REGION Network 7: Choose Flush Destination
   // #Cmd.Flush_Select.%X0 = T-20.00
   // #Cmd.Flush_Select.%X1 = T-21.00
   // #Cmd.Flush_Select.%X2 = T-30.00
   // #Cmd.Flush_Select.%X3 = T-31.00
   // #Cmd.Flush_Select.%X4 = Drain
   // #Cmd.Flush_Select.%X5 = Flush_Selected
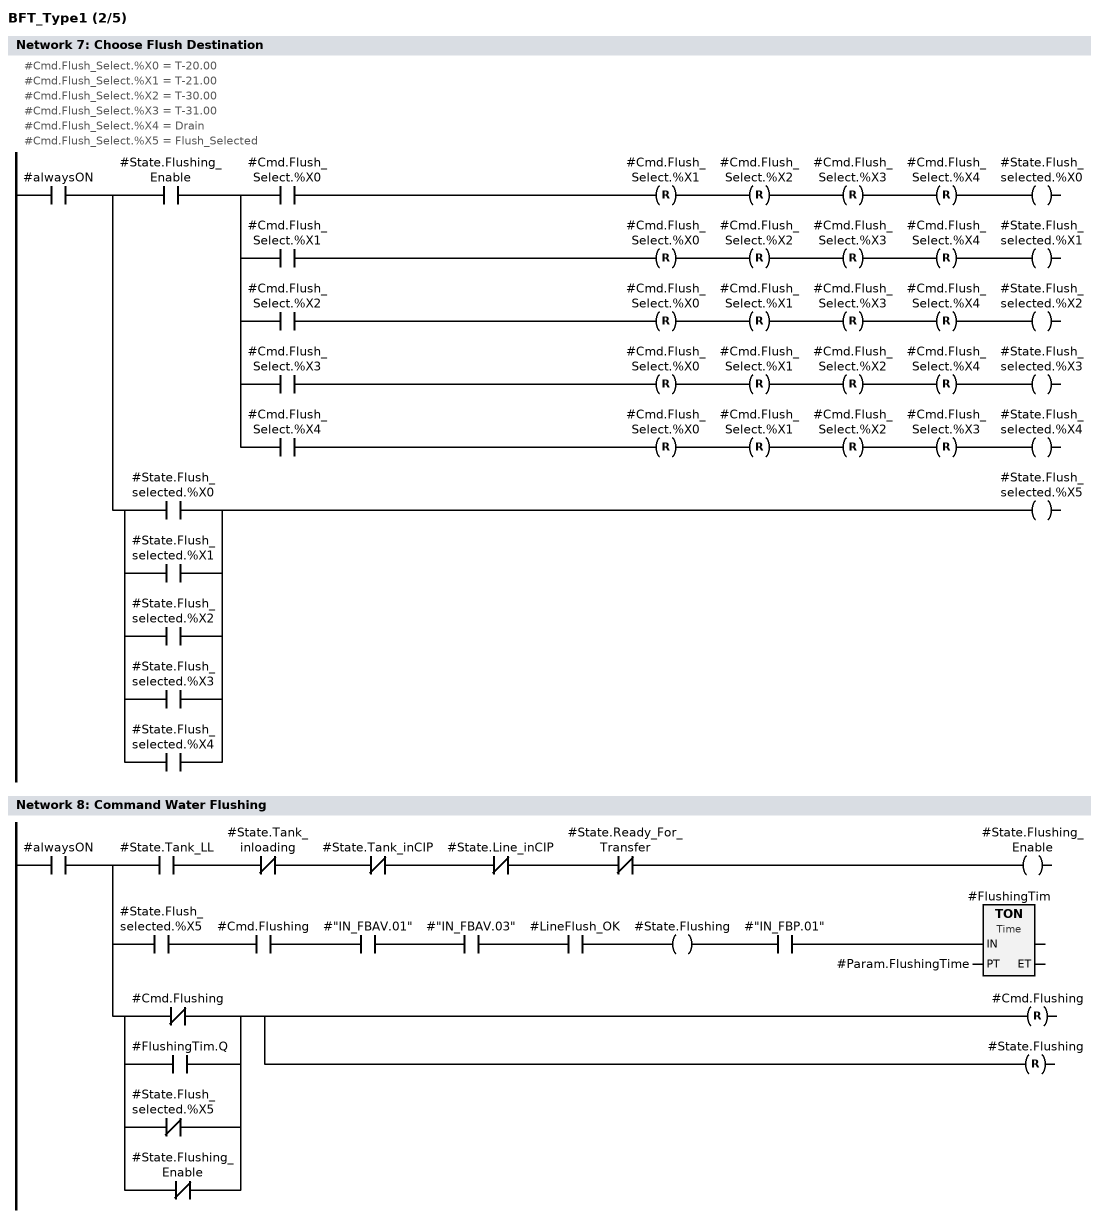
   RUNG wire#powerrail
      Contact( #alwaysON )
      wire#w1
      Contact( #State.Flushing_Enable )
      wire#w2
      Contact( #Cmd.Flush_Select.%X0 )
      R_Coil( #Cmd.Flush_Select.%X1 )
      R_Coil( #Cmd.Flush_Select.%X2 )
      R_Coil( #Cmd.Flush_Select.%X3 )
      R_Coil( #Cmd.Flush_Select.%X4 )
      Coil( #State.Flush_selected.%X0 )
   END_RUNG
   RUNG wire#w2
      Contact( #Cmd.Flush_Select.%X1 )
      R_Coil( #Cmd.Flush_Select.%X0 )
      R_Coil( #Cmd.Flush_Select.%X2 )
      R_Coil( #Cmd.Flush_Select.%X3 )
      R_Coil( #Cmd.Flush_Select.%X4 )
      Coil( #State.Flush_selected.%X1 )
   END_RUNG
   RUNG wire#w2
      Contact( #Cmd.Flush_Select.%X2 )
      R_Coil( #Cmd.Flush_Select.%X0 )
      R_Coil( #Cmd.Flush_Select.%X1 )
      R_Coil( #Cmd.Flush_Select.%X3 )
      R_Coil( #Cmd.Flush_Select.%X4 )
      Coil( #State.Flush_selected.%X2 )
   END_RUNG
   RUNG wire#w2
      Contact( #Cmd.Flush_Select.%X3 )
      R_Coil( #Cmd.Flush_Select.%X0 )
      R_Coil( #Cmd.Flush_Select.%X1 )
      R_Coil( #Cmd.Flush_Select.%X2 )
      R_Coil( #Cmd.Flush_Select.%X4 )
      Coil( #State.Flush_selected.%X3 )
   END_RUNG
   RUNG wire#w2
      Contact( #Cmd.Flush_Select.%X4 )
      R_Coil( #Cmd.Flush_Select.%X0 )
      R_Coil( #Cmd.Flush_Select.%X1 )
      R_Coil( #Cmd.Flush_Select.%X2 )
      R_Coil( #Cmd.Flush_Select.%X3 )
      Coil( #State.Flush_selected.%X4 )
   END_RUNG
   RUNG wire#w1
      Contact( #State.Flush_selected.%X0 )
      wire#w3
      Coil( #State.Flush_selected.%X5 )
   END_RUNG
   RUNG wire#w1
      Contact( #State.Flush_selected.%X1 )
   END_RUNG wire#w3
   RUNG wire#w1
      Contact( #State.Flush_selected.%X2 )
   END_RUNG wire#w3
   RUNG wire#w1
      Contact( #State.Flush_selected.%X3 )
   END_RUNG wire#w3
   RUNG wire#w1
      Contact( #State.Flush_selected.%X4 )
   END_RUNG wire#w3
   // the same network as SCL:
   #_w1 := #alwaysON AND #State.Flushing_Enable;
   #_w2 := #_w1 AND #Cmd.Flush_Select.%X0;
   IF #_w2 THEN
       #Cmd.Flush_Select.%X1 := FALSE;
       #Cmd.Flush_Select.%X2 := FALSE;
       #Cmd.Flush_Select.%X3 := FALSE;
       #Cmd.Flush_Select.%X4 := FALSE;
   END_IF;
   #State.Flush_selected.%X0 := #_w2;
   #_w3 := #_w1 AND #Cmd.Flush_Select.%X1;
   IF #_w3 THEN
       #Cmd.Flush_Select.%X0 := FALSE;
       #Cmd.Flush_Select.%X2 := FALSE;
       #Cmd.Flush_Select.%X3 := FALSE;
       #Cmd.Flush_Select.%X4 := FALSE;
   END_IF;
   #State.Flush_selected.%X1 := #_w3;
   #_w4 := #_w1 AND #Cmd.Flush_Select.%X2;
   IF #_w4 THEN
       #Cmd.Flush_Select.%X0 := FALSE;
       #Cmd.Flush_Select.%X1 := FALSE;
       #Cmd.Flush_Select.%X3 := FALSE;
       #Cmd.Flush_Select.%X4 := FALSE;
   END_IF;
   #State.Flush_selected.%X2 := #_w4;
   #_w5 := #_w1 AND #Cmd.Flush_Select.%X3;
   IF #_w5 THEN
       #Cmd.Flush_Select.%X0 := FALSE;
       #Cmd.Flush_Select.%X1 := FALSE;
       #Cmd.Flush_Select.%X2 := FALSE;
       #Cmd.Flush_Select.%X4 := FALSE;
   END_IF;
   #State.Flush_selected.%X3 := #_w5;
   #_w6 := #_w1 AND #Cmd.Flush_Select.%X4;
   IF #_w6 THEN
       #Cmd.Flush_Select.%X0 := FALSE;
       #Cmd.Flush_Select.%X1 := FALSE;
       #Cmd.Flush_Select.%X2 := FALSE;
       #Cmd.Flush_Select.%X3 := FALSE;
   END_IF;
   #State.Flush_selected.%X4 := #_w6;
   #State.Flush_selected.%X5 := #alwaysON AND (#State.Flush_selected.%X0 OR #State.Flush_selected.%X1 OR #State.Flush_selected.%X2 OR #State.Flush_selected.%X3 OR #State.Flush_selected.%X4);
END_REGION

REGION Network 8: Command Water Flushing
   RUNG wire#powerrail
      Contact( #alwaysON )
      wire#w1
      Contact( #State.Tank_LL )
      I_Contact( #State.Tank_inloading )
      I_Contact( #State.Tank_inCIP )
      I_Contact( #State.Line_inCIP )
      I_Contact( #State.Ready_For_Transfer )
      Coil( #State.Flushing_Enable )
   END_RUNG
   RUNG wire#w1
      Contact( #State.Flush_selected.%X5 )
      Contact( #Cmd.Flushing )
      Contact( #"IN_FBAV.01" )
      Contact( #"IN_FBAV.03" )
      Contact( #LineFlush_OK )
      Coil( #State.Flushing )
      Contact( #"IN_FBP.01" )
      { S7_Templates := "time_type := Time" } #FlushingTim.TON(pt := #Param.FlushingTime, et =>)
   END_RUNG
   RUNG wire#w1
      I_Contact( #Cmd.Flushing )
      wire#w2
      R_Coil( #Cmd.Flushing )
   END_RUNG
   RUNG wire#w1
      Contact( #FlushingTim.Q )
   END_RUNG wire#w2
   RUNG wire#w1
      I_Contact( #State.Flush_selected.%X5 )
   END_RUNG wire#w2
   RUNG wire#w1
      I_Contact( #State.Flushing_Enable )
   END_RUNG wire#w2
   RUNG wire#w2
      R_Coil( #State.Flushing )
   END_RUNG
   // the same network as SCL:
   #State.Flushing_Enable := #alwaysON AND #State.Tank_LL AND NOT #State.Tank_inloading AND NOT #State.Tank_inCIP AND NOT #State.Line_inCIP AND NOT #State.Ready_For_Transfer;
   #State.Flushing := #alwaysON AND #State.Flush_selected.%X5 AND #Cmd.Flushing AND #"IN_FBAV.01" AND #"IN_FBAV.03" AND #LineFlush_OK;
   #FlushingTim(IN := #State.Flushing AND #"IN_FBP.01", PT := #Param.FlushingTime);   // TON
   #_w1 := #alwaysON AND (NOT #Cmd.Flushing OR #FlushingTim.Q OR NOT #State.Flush_selected.%X5 OR NOT #State.Flushing_Enable);
   IF #_w1 THEN
       #Cmd.Flushing := FALSE;
       #State.Flushing := FALSE;
   END_IF;
END_REGION

REGION Network 9: Flushing Destination AV and Pump
   // #Cmd.Flush_Select.%X0 = T-20.00
   // #Cmd.Flush_Select.%X1 = T-21.00
   // #Cmd.Flush_Select.%X2 = T-30.00
   // #Cmd.Flush_Select.%X3 = T-31.00
   // #Cmd.Flush_Select.%X4 = Drain
   // #Cmd.Flush_Select.%X5 = Flush_Selected
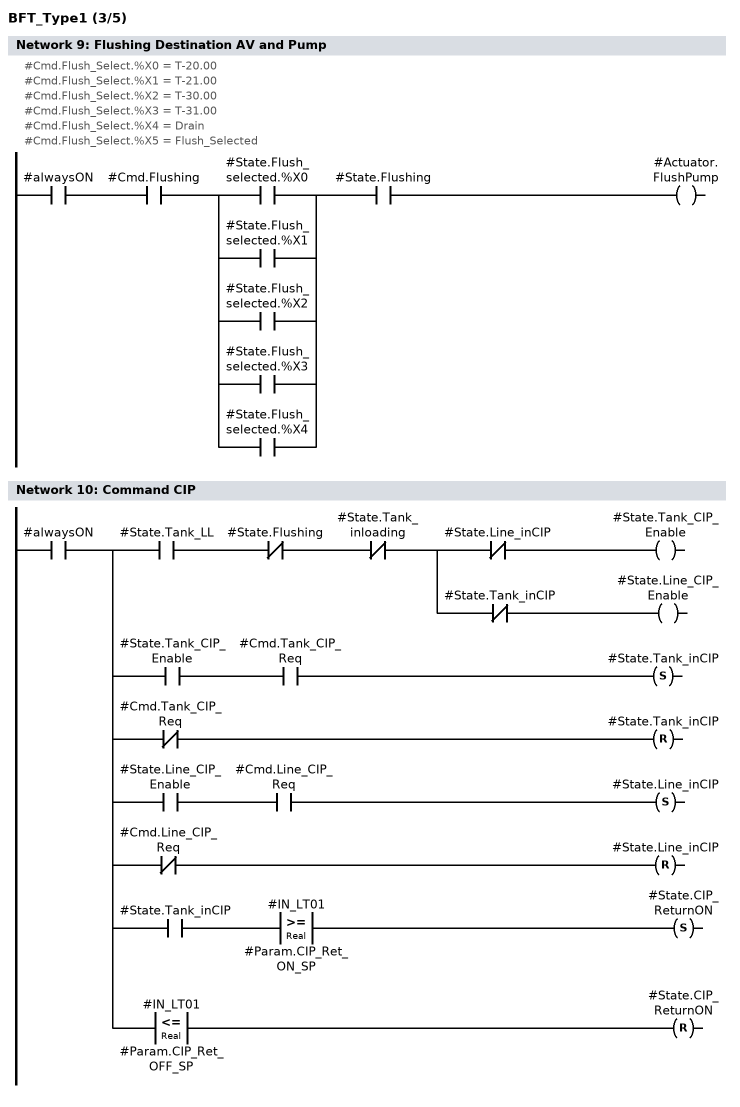
   RUNG wire#powerrail
      Contact( #alwaysON )
      Contact( #Cmd.Flushing )
      wire#w1
      Contact( #State.Flush_selected.%X0 )
      wire#w2
      Contact( #State.Flushing )
      Coil( #Actuator.FlushPump )
   END_RUNG
   RUNG wire#w1
      Contact( #State.Flush_selected.%X1 )
   END_RUNG wire#w2
   RUNG wire#w1
      Contact( #State.Flush_selected.%X2 )
   END_RUNG wire#w2
   RUNG wire#w1
      Contact( #State.Flush_selected.%X3 )
   END_RUNG wire#w2
   RUNG wire#w1
      Contact( #State.Flush_selected.%X4 )
   END_RUNG wire#w2
   // the same network as SCL:
   #Actuator.FlushPump := #alwaysON AND #Cmd.Flushing AND (#State.Flush_selected.%X0 OR #State.Flush_selected.%X1 OR #State.Flush_selected.%X2 OR #State.Flush_selected.%X3 OR #State.Flush_selected.%X4) AND #State.Flushing;
END_REGION

REGION Network 10: Command CIP
   RUNG wire#powerrail
      Contact( #alwaysON )
      wire#w1
      Contact( #State.Tank_LL )
      I_Contact( #State.Flushing )
      I_Contact( #State.Tank_inloading )
      wire#w2
      I_Contact( #State.Line_inCIP )
      Coil( #State.Tank_CIP_Enable )
   END_RUNG
   RUNG wire#w2
      I_Contact( #State.Tank_inCIP )
      Coil( #State.Line_CIP_Enable )
   END_RUNG
   RUNG wire#w1
      Contact( #State.Tank_CIP_Enable )
      Contact( #Cmd.Tank_CIP_Req )
      S_Coil( #State.Tank_inCIP )
   END_RUNG
   RUNG wire#w1
      I_Contact( #Cmd.Tank_CIP_Req )
      R_Coil( #State.Tank_inCIP )
   END_RUNG
   RUNG wire#w1
      Contact( #State.Line_CIP_Enable )
      Contact( #Cmd.Line_CIP_Req )
      S_Coil( #State.Line_inCIP )
   END_RUNG
   RUNG wire#w1
      I_Contact( #Cmd.Line_CIP_Req )
      R_Coil( #State.Line_inCIP )
   END_RUNG
   RUNG wire#w1
      Contact( #State.Tank_inCIP )
      { S7_Templates := "SrcType := Real" } GE_Contact(in1 := #IN_LT01, in2 := #Param.CIP_Ret_ON_SP)
      S_Coil( #State.CIP_ReturnON )
   END_RUNG
   RUNG wire#w1
      { S7_Templates := "SrcType := Real" } LE_Contact(in1 := #IN_LT01, in2 := #Param.CIP_Ret_OFF_SP)
      R_Coil( #State.CIP_ReturnON )
   END_RUNG
   // the same network as SCL:
   #_w1 := #alwaysON AND #State.Tank_LL AND NOT #State.Flushing AND NOT #State.Tank_inloading;
   #State.Tank_CIP_Enable := #_w1 AND NOT #State.Line_inCIP;
   #State.Line_CIP_Enable := #_w1 AND NOT #State.Tank_inCIP;
   IF #alwaysON AND #State.Tank_CIP_Enable AND #Cmd.Tank_CIP_Req THEN #State.Tank_inCIP := TRUE; END_IF;
   IF #alwaysON AND NOT #Cmd.Tank_CIP_Req THEN #State.Tank_inCIP := FALSE; END_IF;
   IF #alwaysON AND #State.Line_CIP_Enable AND #Cmd.Line_CIP_Req THEN #State.Line_inCIP := TRUE; END_IF;
   IF #alwaysON AND NOT #Cmd.Line_CIP_Req THEN #State.Line_inCIP := FALSE; END_IF;
   IF #alwaysON AND #State.Tank_inCIP AND (#IN_LT01 >= #Param.CIP_Ret_ON_SP) THEN
       #State.CIP_ReturnON := TRUE;
   END_IF;
   IF #alwaysON AND (#IN_LT01 <= #Param.CIP_Ret_OFF_SP) THEN #State.CIP_ReturnON := FALSE; END_IF;
END_REGION

REGION Network 11: Loading AV and Pump
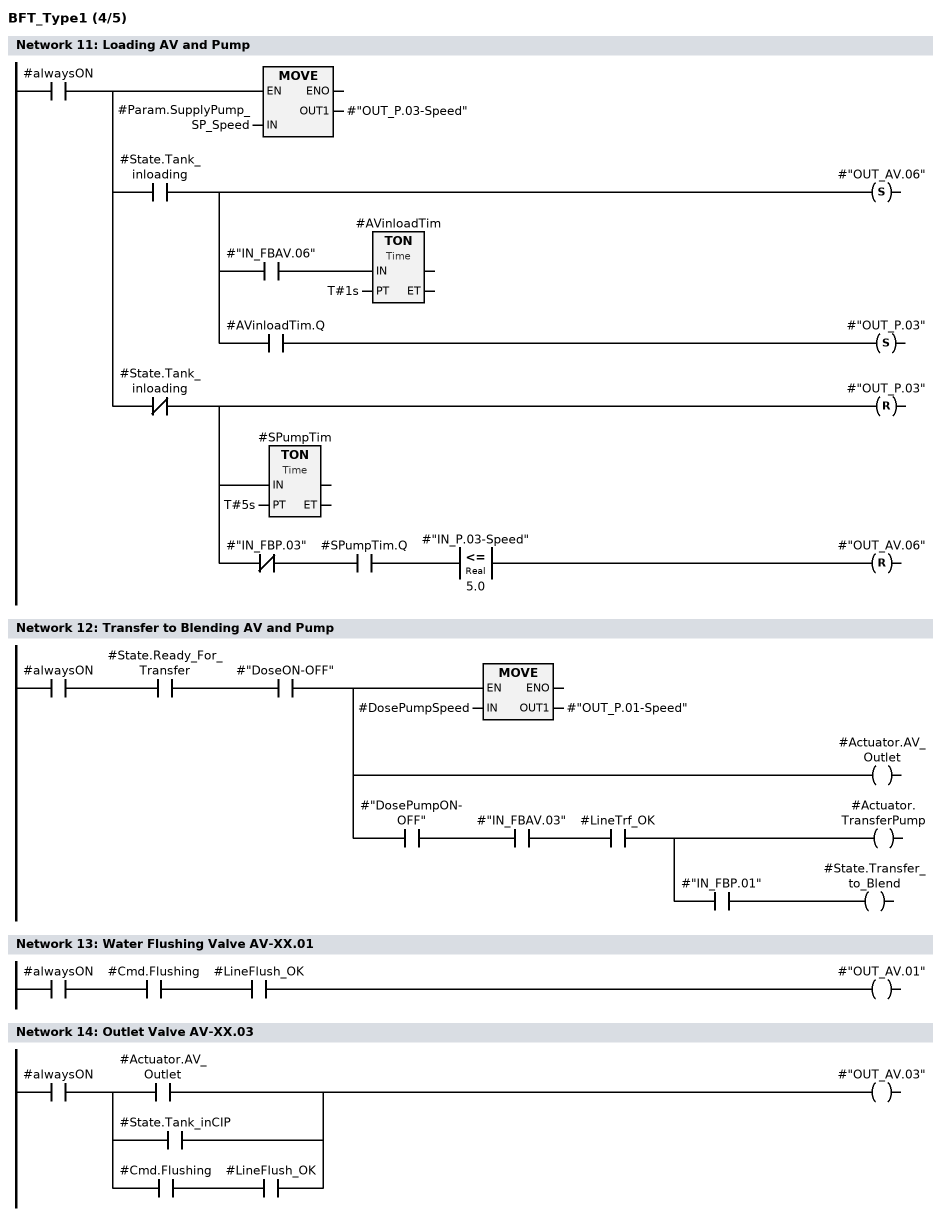
   RUNG wire#powerrail
      Contact( #alwaysON )
      wire#w1
      Move(in := #Param.SupplyPump_SP_Speed, out1 => #"OUT_P.03-Speed")
   END_RUNG
   RUNG wire#w1
      Contact( #State.Tank_inloading )
      wire#w2
      S_Coil( #"OUT_AV.06" )
   END_RUNG
   RUNG wire#w2
      Contact( #"IN_FBAV.06" )
      { S7_Templates := "time_type := Time" } #AVinloadTim.TON(pt := T#1s, et =>)
   END_RUNG
   RUNG wire#w2
      Contact( #AVinloadTim.Q )
      S_Coil( #"OUT_P.03" )
   END_RUNG
   RUNG wire#w1
      I_Contact( #State.Tank_inloading )
      wire#w3
      R_Coil( #"OUT_P.03" )
   END_RUNG
   RUNG wire#w3
      { S7_Templates := "time_type := Time" } #SPumpTim.TON(pt := T#5s, et =>)
   END_RUNG
   RUNG wire#w3
      I_Contact( #"IN_FBP.03" )
      Contact( #SPumpTim.Q )
      { S7_Templates := "SrcType := Real" } LE_Contact(in1 := #"IN_P.03-Speed", in2 := 5.0)
      R_Coil( #"OUT_AV.06" )
   END_RUNG
   // the same network as SCL:
   IF #alwaysON THEN #"OUT_P.03-Speed" := #Param.SupplyPump_SP_Speed; END_IF;
   #_w1 := #alwaysON AND #State.Tank_inloading;
   IF #_w1 THEN #"OUT_AV.06" := TRUE; END_IF;
   #AVinloadTim(IN := #_w1 AND #"IN_FBAV.06", PT := T#1s);   // TON
   IF #_w1 AND #AVinloadTim.Q THEN #"OUT_P.03" := TRUE; END_IF;
   #_w2 := #alwaysON AND NOT #State.Tank_inloading;
   IF #_w2 THEN #"OUT_P.03" := FALSE; END_IF;
   #SPumpTim(IN := #_w2, PT := T#5s);   // TON
   IF #_w2 AND NOT #"IN_FBP.03" AND #SPumpTim.Q AND (#"IN_P.03-Speed" <= 5.0) THEN
       #"OUT_AV.06" := FALSE;
   END_IF;
END_REGION

REGION Network 12: Transfer to Blending AV and Pump
   RUNG wire#powerrail
      Contact( #alwaysON )
      Contact( #State.Ready_For_Transfer )
      Contact( #"DoseON-OFF" )
      wire#w1
      Move(in := #DosePumpSpeed, out1 => #"OUT_P.01-Speed")
   END_RUNG
   RUNG wire#w1
      Coil( #Actuator.AV_Outlet )
   END_RUNG
   RUNG wire#w1
      Contact( #"DosePumpON-OFF" )
      Contact( #"IN_FBAV.03" )
      Contact( #LineTrf_OK )
      wire#w2
      Coil( #Actuator.TransferPump )
   END_RUNG
   RUNG wire#w2
      Contact( #"IN_FBP.01" )
      Coil( #State.Transfer_to_Blend )
   END_RUNG
   // the same network as SCL:
   #_w1 := #alwaysON AND #State.Ready_For_Transfer AND #"DoseON-OFF";
   IF #_w1 THEN #"OUT_P.01-Speed" := #DosePumpSpeed; END_IF;
   #Actuator.AV_Outlet := #_w1;
   #Actuator.TransferPump := #_w1 AND #"DosePumpON-OFF" AND #"IN_FBAV.03" AND #LineTrf_OK;
   #State.Transfer_to_Blend := #Actuator.TransferPump AND #"IN_FBP.01";
END_REGION

REGION Network 13: Water Flushing Valve AV-XX.01
   RUNG wire#powerrail
      Contact( #alwaysON )
      Contact( #Cmd.Flushing )
      Contact( #LineFlush_OK )
      Coil( #"OUT_AV.01" )
   END_RUNG
   // the same network as SCL:
   #"OUT_AV.01" := #alwaysON AND #Cmd.Flushing AND #LineFlush_OK;
END_REGION

REGION Network 14: Outlet Valve AV-XX.03
   RUNG wire#powerrail
      Contact( #alwaysON )
      wire#w1
      Contact( #Actuator.AV_Outlet )
      wire#w2
      Coil( #"OUT_AV.03" )
   END_RUNG
   RUNG wire#w1
      Contact( #State.Tank_inCIP )
   END_RUNG wire#w2
   RUNG wire#w1
      Contact( #Cmd.Flushing )
      Contact( #LineFlush_OK )
   END_RUNG wire#w2
   // the same network as SCL:
   #"OUT_AV.03" := #alwaysON AND (#Actuator.AV_Outlet OR #State.Tank_inCIP OR (#Cmd.Flushing AND #LineFlush_OK));
END_REGION

REGION Network 15: CIP Valve AV-XX.02, 04, 07
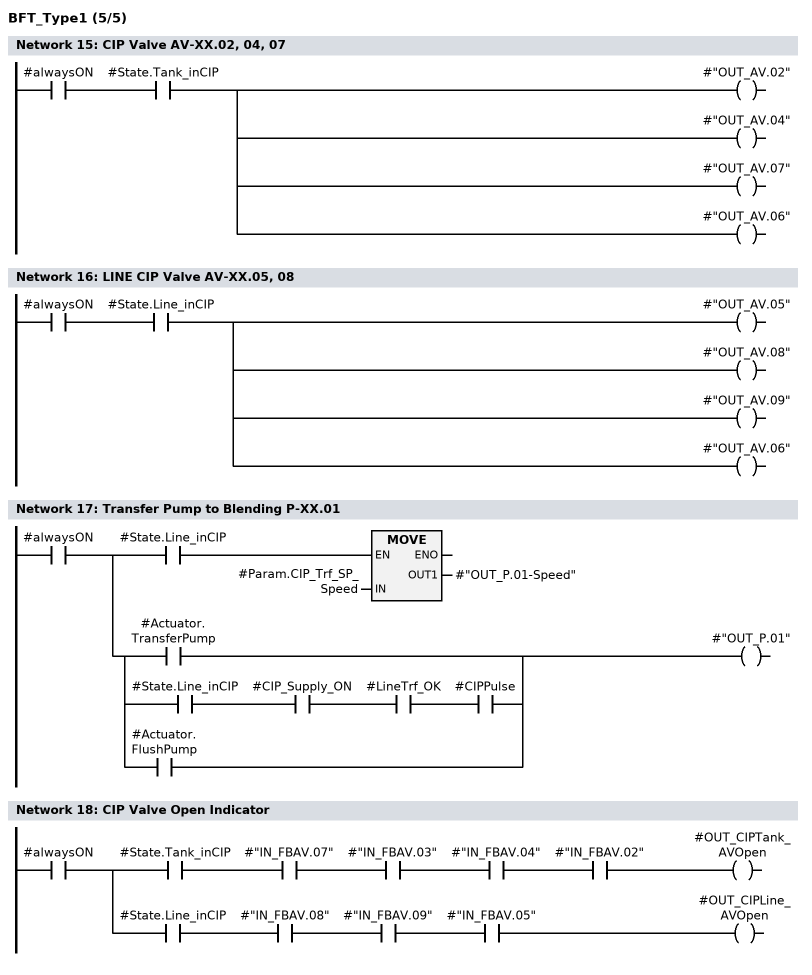
   RUNG wire#powerrail
      Contact( #alwaysON )
      Contact( #State.Tank_inCIP )
      wire#w1
      Coil( #"OUT_AV.02" )
   END_RUNG
   RUNG wire#w1
      Coil( #"OUT_AV.04" )
   END_RUNG
   RUNG wire#w1
      Coil( #"OUT_AV.07" )
   END_RUNG
   RUNG wire#w1
      Coil( #"OUT_AV.06" )
   END_RUNG
   // the same network as SCL:
   #"OUT_AV.02" := #alwaysON AND #State.Tank_inCIP;
   #"OUT_AV.04" := #"OUT_AV.02";
   #"OUT_AV.07" := #"OUT_AV.02";
   #"OUT_AV.06" := #"OUT_AV.02";
END_REGION

REGION Network 16: LINE CIP Valve AV-XX.05, 08
   RUNG wire#powerrail
      Contact( #alwaysON )
      Contact( #State.Line_inCIP )
      wire#w1
      Coil( #"OUT_AV.05" )
   END_RUNG
   RUNG wire#w1
      Coil( #"OUT_AV.08" )
   END_RUNG
   RUNG wire#w1
      Coil( #"OUT_AV.09" )
   END_RUNG
   RUNG wire#w1
      Coil( #"OUT_AV.06" )
   END_RUNG
   // the same network as SCL:
   #"OUT_AV.05" := #alwaysON AND #State.Line_inCIP;
   #"OUT_AV.08" := #"OUT_AV.05";
   #"OUT_AV.09" := #"OUT_AV.05";
   #"OUT_AV.06" := #"OUT_AV.05";
END_REGION

REGION Network 17: Transfer Pump to Blending P-XX.01
   RUNG wire#powerrail
      Contact( #alwaysON )
      wire#w1
      Contact( #State.Line_inCIP )
      Move(in := #Param.CIP_Trf_SP_Speed, out1 => #"OUT_P.01-Speed")
   END_RUNG
   RUNG wire#w1
      Contact( #Actuator.TransferPump )
      wire#w2
      Coil( #"OUT_P.01" )
   END_RUNG
   RUNG wire#w1
      Contact( #State.Line_inCIP )
      Contact( #CIP_Supply_ON )
      Contact( #LineTrf_OK )
      Contact( #CIPPulse )
   END_RUNG wire#w2
   RUNG wire#w1
      Contact( #Actuator.FlushPump )
   END_RUNG wire#w2
   // the same network as SCL:
   IF #alwaysON AND #State.Line_inCIP THEN #"OUT_P.01-Speed" := #Param.CIP_Trf_SP_Speed; END_IF;
   #"OUT_P.01" := #alwaysON AND (#Actuator.TransferPump OR (#State.Line_inCIP AND #CIP_Supply_ON AND #LineTrf_OK AND #CIPPulse) OR #Actuator.FlushPump);
END_REGION

REGION Network 18: CIP Valve Open Indicator
   RUNG wire#powerrail
      Contact( #alwaysON )
      wire#w1
      Contact( #State.Tank_inCIP )
      Contact( #"IN_FBAV.07" )
      Contact( #"IN_FBAV.03" )
      Contact( #"IN_FBAV.04" )
      Contact( #"IN_FBAV.02" )
      Coil( #OUT_CIPTank_AVOpen )
   END_RUNG
   RUNG wire#w1
      Contact( #State.Line_inCIP )
      Contact( #"IN_FBAV.08" )
      Contact( #"IN_FBAV.09" )
      Contact( #"IN_FBAV.05" )
      Coil( #OUT_CIPLine_AVOpen )
   END_RUNG
   // the same network as SCL:
   #OUT_CIPTank_AVOpen := #alwaysON AND #State.Tank_inCIP AND #"IN_FBAV.07" AND #"IN_FBAV.03" AND #"IN_FBAV.04" AND #"IN_FBAV.02";
   #OUT_CIPLine_AVOpen := #alwaysON AND #State.Line_inCIP AND #"IN_FBAV.08" AND #"IN_FBAV.09" AND #"IN_FBAV.05";
END_REGION
END_FUNCTION_BLOCK

FUNCTION_BLOCK "BFT_Type3"   // FB353, LAD
{ S7_Optimized_Access := 'TRUE' }
VERSION : 0.1
// Buffer Tank Chili Fresh
// stored: AutoNumber false, IsIECCheckEnabled false, IsRetainMemResEnabled false, MemoryReserve 100, SetENOAutomatically false, UDAEnableTagReadback false
   VAR_INPUT
      "IN_FBAV.01" : Bool := FALSE;   // Tank Flushing Water Valve
      "IN_FBAV.02" : Bool := FALSE;   // Tank CIP Top Inlet Valve
      "IN_FBAV.03" : Bool := FALSE;   // Tank Tank Outlet Valve
      "IN_FBAV.04" : Bool := FALSE;   // Tank CIP Return Valve
      "IN_FBAV.05" : Bool := FALSE;   // Line CIP Bypass Valve
      "IN_FBAV.06" : Bool := FALSE;   // Tank CIP Valve
      "IN_FBAV.11" : Bool;   // Line CIP Valve
      "IN_FBAV.12" : Bool := FALSE;   // Line CIP Valve
      IN_LT01 : Real;   // Tank Level Transmitter
      "IN_FBP.01" : Bool := FALSE;   // Transfer Pump
      "IN_P.01-Speed" : Real;   // Transfer Pump AV Speed
      "IN_FBP.02" : Bool := FALSE;   // CIP Pump
      "IN_P.02-Speed" : Real;   // CIP Pump AV Speed
      "IN_FBP.03" : Bool := FALSE;   // Supply Pump
      "IN_P.03-Speed" : Real;   // Supply Pump AV Speed
      DosePumpSpeed : Real;
      "DoseON-OFF" : Bool := FALSE;
      "DosePumpON-OFF" : Bool := FALSE;
      CIPPulse : Bool := FALSE;
      CIP_Supply_ON : Bool;
      LineTrf_OK : Bool := FALSE;
      LineFlush_OK : Bool;
      Loading_Busy : Bool;   // Other tank at loading
   END_VAR
   VAR_OUTPUT
      "OUT_AV.01" : Bool := FALSE;   // Tank Flushing Water Valve
      "OUT_AV.02" : Bool := FALSE;   // Tank CIP Top Inlet Valve
      "OUT_AV.03" : Bool := FALSE;   // Tank Tank Outlet Valve
      "OUT_AV.04" : Bool := FALSE;   // Tank CIP Return Valve
      "OUT_AV.05" : Bool := FALSE;   // Line CIP Bypass Valve
      "OUT_AV.06" : Bool := FALSE;   // Tank CIP Valve
      OUT_Inload : Bool := FALSE;
      "OUT_AV.11" : Bool;   // Line CIP Valve
      "OUT_AV.12" : Bool := FALSE;   // Line CIP Valve
      "OUT_P.01" : Bool := FALSE;   // Transfer Pump
      "OUT_P.01-Speed" : Real;   // Transfer Pump AV Speed
      "OUT_P.02" : Bool := FALSE;   // CIP Pump
      "OUT_P.02-Speed" : Real;   // CIP Pump AV Speed
      "OUT_P.03" : Bool := FALSE;   // Supply Pump
      "OUT_P.03-Speed" : Real;   // Supply Pump AV Speed
      OUT_CIPTank_AVOpen : Bool;
      OUT_CIPLine_AVOpen : Bool;
   END_VAR
   VAR
      Cmd { ExternalAccessible := 'False'; ExternalVisible := 'False'; ExternalWritable := 'False'} : Struct
         Inload { ExternalAccessible := 'False'; ExternalVisible := 'False'; ExternalWritable := 'False'} : Bool;   // Start Loading
         Tank_CIP_Req { ExternalAccessible := 'False'; ExternalVisible := 'False'; ExternalWritable := 'False'} : Bool;
         Line_CIP_Req { ExternalAccessible := 'False'; ExternalVisible := 'False'; ExternalWritable := 'False'} : Bool;
         Flushing { ExternalAccessible := 'False'; ExternalVisible := 'False'; ExternalWritable := 'False'} : Bool;   // Water Flushing
         Flush_Select { ExternalAccessible := 'False'; ExternalVisible := 'False'; ExternalWritable := 'False'} : Byte;
         RaadyForMix { ExternalAccessible := 'False'; ExternalVisible := 'False'; ExternalWritable := 'False'} : Bool;   // Tank Ready for Blending
      END_STRUCT;
      Param { ExternalAccessible := 'False'; ExternalVisible := 'False'; ExternalWritable := 'False'} : Struct
         SP_Level_LL { ExternalAccessible := 'False'; ExternalVisible := 'False'; ExternalWritable := 'False'} : Real := 10.0;
         SP_Level_ML { ExternalAccessible := 'False'; ExternalVisible := 'False'; ExternalWritable := 'False'} : Real := 80.0;
         SP_Level_HL { ExternalAccessible := 'False'; ExternalVisible := 'False'; ExternalWritable := 'False'} : Real := 100.0;
         SupplyPump_SP_Speed { ExternalAccessible := 'False'; ExternalVisible := 'False'; ExternalWritable := 'False'} : Real := 80.0;
         L_Hi_Lim { ExternalAccessible := 'False'; ExternalVisible := 'False'; ExternalWritable := 'False'} : Real := 100.0;
         L_Lo_Lim { ExternalAccessible := 'False'; ExternalVisible := 'False'; ExternalWritable := 'False'} : Real := 0.0;
         L_Hys { ExternalAccessible := 'False'; ExternalVisible := 'False'; ExternalWritable := 'False'} : Real := 5.0;
         FlushingTime { ExternalAccessible := 'False'; ExternalVisible := 'False'; ExternalWritable := 'False'} : Time := T#10s;
         CIP_Trf_SP_Speed { ExternalAccessible := 'False'; ExternalVisible := 'False'; ExternalWritable := 'False'} : Real := 80.0;
         CIP_Ret_ON_SP { ExternalAccessible := 'False'; ExternalVisible := 'False'; ExternalWritable := 'False'} : Real := 5.0;
         CIP_Ret_OFF_SP { ExternalAccessible := 'False'; ExternalVisible := 'False'; ExternalWritable := 'False'} : Real;
      END_STRUCT;
      State { ExternalAccessible := 'False'; ExternalVisible := 'False'; ExternalWritable := 'False'} : Struct   // Tank in loading state
         Tank_inloading { ExternalAccessible := 'False'; ExternalVisible := 'False'; ExternalWritable := 'False'} : Bool;
         Tank_inCIP { ExternalAccessible := 'False'; ExternalVisible := 'False'; ExternalWritable := 'False'} : Bool;
         Line_inCIP { ExternalAccessible := 'False'; ExternalVisible := 'False'; ExternalWritable := 'False'} : Bool;
         Flushing { ExternalAccessible := 'False'; ExternalVisible := 'False'; ExternalWritable := 'False'} : Bool;
         Tank_LL { ExternalAccessible := 'False'; ExternalVisible := 'False'; ExternalWritable := 'False'} : Bool;
         Tank_ML { ExternalAccessible := 'False'; ExternalVisible := 'False'; ExternalWritable := 'False'} : Bool;
         Tank_HL { ExternalAccessible := 'False'; ExternalVisible := 'False'; ExternalWritable := 'False'} : Bool;
         Inload_Enable { ExternalAccessible := 'False'; ExternalVisible := 'False'; ExternalWritable := 'False'} : Bool;
         Tank_CIP_Enable { ExternalAccessible := 'False'; ExternalVisible := 'False'; ExternalWritable := 'False'} : Bool;
         Line_CIP_Enable { ExternalAccessible := 'False'; ExternalVisible := 'False'; ExternalWritable := 'False'} : Bool;
         Flushing_Enable { ExternalAccessible := 'False'; ExternalVisible := 'False'; ExternalWritable := 'False'} : Bool;
         Flush_selected { ExternalAccessible := 'False'; ExternalVisible := 'False'; ExternalWritable := 'False'} : Byte;
         CIP_Request_OK { ExternalAccessible := 'False'; ExternalVisible := 'False'; ExternalWritable := 'False'} : Bool;
         CIP_ReturnON { ExternalAccessible := 'False'; ExternalVisible := 'False'; ExternalWritable := 'False'} : Bool;
         Ready_For_Transfer_EN { ExternalAccessible := 'False'; ExternalVisible := 'False'; ExternalWritable := 'False'} : Bool;   // Tank Ready for Transfer to Blending
         Ready_For_Transfer { ExternalAccessible := 'False'; ExternalVisible := 'False'; ExternalWritable := 'False'} : Bool;   // Tank Ready for Transfer to Blending
         Transfer_to_Blend { ExternalAccessible := 'False'; ExternalVisible := 'False'; ExternalWritable := 'False'} : Bool;
         HWT_Status { ExternalAccessible := 'False'; ExternalVisible := 'False'; ExternalWritable := 'False'} : Int;
      END_STRUCT;
      alwaysON : Bool;
      L_Hys_Abs : Real;
      Hys_Level_HL : Real;
      Hys_Level_ML : Real;
      Hys_Level_LL : Real;
      r : Struct
         PosE1 : Bool;
         PosE2 : Bool;
         PosE3 : Bool;
         PosE4 : Bool;
         PosE5 : Bool;
         PosE6 : Bool;
         PosE7 : Bool;
         PosE8 : Bool;
         PosE9 : Bool;
         PosE10 : Bool;
         PosE11 : Bool;
         PosE12 : Bool;
         PosE13 : Bool;
         PosE14 : Bool;
         PosE15 : Bool;
         PosE16 : Bool;
         PosE17 : Bool;
         PosE18 : Bool;
         PosE19 : Bool;
         PosE20 : Bool;
         PosE21 : Bool;
         PosE22 : Bool;
         PosE23 : Bool;
         PosE24 : Bool;
         PosE25 : Bool;
         PosE26 : Bool;
         PosE27 : Bool;
         PosE28 : Bool;
         PosE29 : Bool;
         PosE30 : Bool;
         PosE31 : Bool;
         PosE32 : Bool;
      END_STRUCT;
      Actuator : Struct
         AV_Outlet : Bool;
         TransferPump : Bool;
         FlushPump : Bool;
         CV_Steam : Bool;
         Pump : Bool;
      END_STRUCT;
      FlushingTim : TON_TIME;
      SPumpTim { S7_SetPoint := 'True'} : TON_TIME;
      AVinloadTim { S7_SetPoint := 'True'} : TON_TIME;
   END_VAR
   VAR_TEMP   // added for the SCL form of the ladder/FBD networks
      _w1 : Bool;
      _w2 : Bool;
      _w3 : Bool;
      _w4 : Bool;
      _w5 : Bool;
      _w6 : Bool;
   END_VAR
BEGIN

REGION Network 1: Always_ON
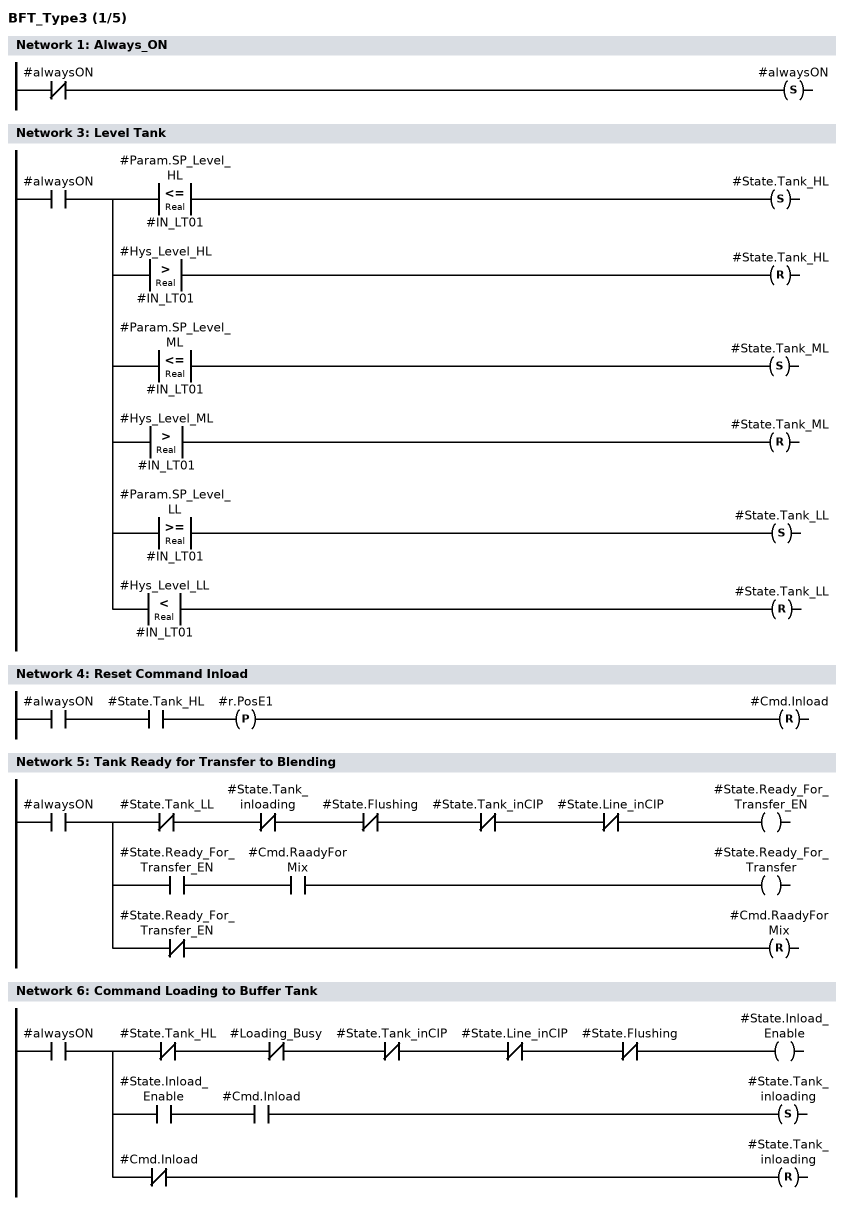
   RUNG wire#powerrail
      I_Contact( #alwaysON )
      S_Coil( #alwaysON )
   END_RUNG
   // the same network as SCL:
   IF NOT #alwaysON THEN #alwaysON := TRUE; END_IF;
END_REGION

NETWORK
TITLE = Hys Calculation
//Level Hys Absolute
      L     #Param.L_Hi_Lim;
      L     #Param.L_Lo_Lim;
      -R;
      L     100.0;
      /R;
      L     #Param.L_Hys;
      *R;
      T     #L_Hys_Abs;
//Tank High Level
      L     #Param.SP_Level_HL;
      L     #L_Hys_Abs;
      -R;
      T     #Hys_Level_HL;
//Tank Mid Level
      L     #Param.SP_Level_ML;
      L     #L_Hys_Abs;
      -R;
      T     #Hys_Level_ML;
//Tank Low Level
      L     #Param.SP_Level_LL;
      L     #L_Hys_Abs;
      +R;
      T     #Hys_Level_LL;


REGION Network 3: Level Tank
   RUNG wire#powerrail
      Contact( #alwaysON )
      wire#w1
      { S7_Templates := "SrcType := Real" } LE_Contact(in1 := #Param.SP_Level_HL, in2 := #IN_LT01)
      S_Coil( #State.Tank_HL )
   END_RUNG
   RUNG wire#w1
      { S7_Templates := "SrcType := Real" } GT_Contact(in1 := #Hys_Level_HL, in2 := #IN_LT01)
      R_Coil( #State.Tank_HL )
   END_RUNG
   RUNG wire#w1
      { S7_Templates := "SrcType := Real" } LE_Contact(in1 := #Param.SP_Level_ML, in2 := #IN_LT01)
      S_Coil( #State.Tank_ML )
   END_RUNG
   RUNG wire#w1
      { S7_Templates := "SrcType := Real" } GT_Contact(in1 := #Hys_Level_ML, in2 := #IN_LT01)
      R_Coil( #State.Tank_ML )
   END_RUNG
   RUNG wire#w1
      { S7_Templates := "SrcType := Real" } GE_Contact(in1 := #Param.SP_Level_LL, in2 := #IN_LT01)
      S_Coil( #State.Tank_LL )
   END_RUNG
   RUNG wire#w1
      { S7_Templates := "SrcType := Real" } LT_Contact(in1 := #Hys_Level_LL, in2 := #IN_LT01)
      R_Coil( #State.Tank_LL )
   END_RUNG
   // the same network as SCL:
   IF #alwaysON AND (#Param.SP_Level_HL <= #IN_LT01) THEN #State.Tank_HL := TRUE; END_IF;
   IF #alwaysON AND (#Hys_Level_HL > #IN_LT01) THEN #State.Tank_HL := FALSE; END_IF;
   IF #alwaysON AND (#Param.SP_Level_ML <= #IN_LT01) THEN #State.Tank_ML := TRUE; END_IF;
   IF #alwaysON AND (#Hys_Level_ML > #IN_LT01) THEN #State.Tank_ML := FALSE; END_IF;
   IF #alwaysON AND (#Param.SP_Level_LL >= #IN_LT01) THEN #State.Tank_LL := TRUE; END_IF;
   IF #alwaysON AND (#Hys_Level_LL < #IN_LT01) THEN #State.Tank_LL := FALSE; END_IF;
END_REGION

REGION Network 4: Reset Command Inload
   RUNG wire#powerrail
      Contact( #alwaysON )
      Contact( #State.Tank_HL )
      P_Trig( #r.PosE1 )
      R_Coil( #Cmd.Inload )
   END_RUNG
   // the same network as SCL:
   #_w1 := #alwaysON AND #State.Tank_HL;
   #_w2 := #_w1 AND NOT #r.PosE1;   // rising edge
   #r.PosE1 := #_w1;
   IF #_w2 THEN #Cmd.Inload := FALSE; END_IF;
END_REGION

REGION Network 5: Tank Ready for Transfer to Blending
   RUNG wire#powerrail
      Contact( #alwaysON )
      wire#w1
      I_Contact( #State.Tank_LL )
      I_Contact( #State.Tank_inloading )
      I_Contact( #State.Flushing )
      I_Contact( #State.Tank_inCIP )
      I_Contact( #State.Line_inCIP )
      Coil( #State.Ready_For_Transfer_EN )
   END_RUNG
   RUNG wire#w1
      Contact( #State.Ready_For_Transfer_EN )
      Contact( #Cmd.RaadyForMix )
      Coil( #State.Ready_For_Transfer )
   END_RUNG
   RUNG wire#w1
      I_Contact( #State.Ready_For_Transfer_EN )
      R_Coil( #Cmd.RaadyForMix )
   END_RUNG
   // the same network as SCL:
   #State.Ready_For_Transfer_EN := #alwaysON AND NOT #State.Tank_LL AND NOT #State.Tank_inloading AND NOT #State.Flushing AND NOT #State.Tank_inCIP AND NOT #State.Line_inCIP;
   #State.Ready_For_Transfer := #alwaysON AND #State.Ready_For_Transfer_EN AND #Cmd.RaadyForMix;
   IF #alwaysON AND NOT #State.Ready_For_Transfer_EN THEN #Cmd.RaadyForMix := FALSE; END_IF;
END_REGION

REGION Network 6: Command Loading to Buffer Tank
   RUNG wire#powerrail
      Contact( #alwaysON )
      wire#w1
      I_Contact( #State.Tank_HL )
      I_Contact( #Loading_Busy )
      I_Contact( #State.Tank_inCIP )
      I_Contact( #State.Line_inCIP )
      I_Contact( #State.Flushing )
      Coil( #State.Inload_Enable )
   END_RUNG
   RUNG wire#w1
      Contact( #State.Inload_Enable )
      Contact( #Cmd.Inload )
      S_Coil( #State.Tank_inloading )
   END_RUNG
   RUNG wire#w1
      I_Contact( #Cmd.Inload )
      R_Coil( #State.Tank_inloading )
   END_RUNG
   // the same network as SCL:
   #State.Inload_Enable := #alwaysON AND NOT #State.Tank_HL AND NOT #Loading_Busy AND NOT #State.Tank_inCIP AND NOT #State.Line_inCIP AND NOT #State.Flushing;
   IF #alwaysON AND #State.Inload_Enable AND #Cmd.Inload THEN #State.Tank_inloading := TRUE; END_IF;
   IF #alwaysON AND NOT #Cmd.Inload THEN #State.Tank_inloading := FALSE; END_IF;
END_REGION

REGION Network 7: Choose Flush Destination
   // #Cmd.Flush_Select.%X0 = T-20.00
   // #Cmd.Flush_Select.%X1 = T-21.00
   // #Cmd.Flush_Select.%X2 = T-30.00
   // #Cmd.Flush_Select.%X3 = T-31.00
   // #Cmd.Flush_Select.%X4 = Drain
   // #Cmd.Flush_Select.%X5 = Flush_Selected
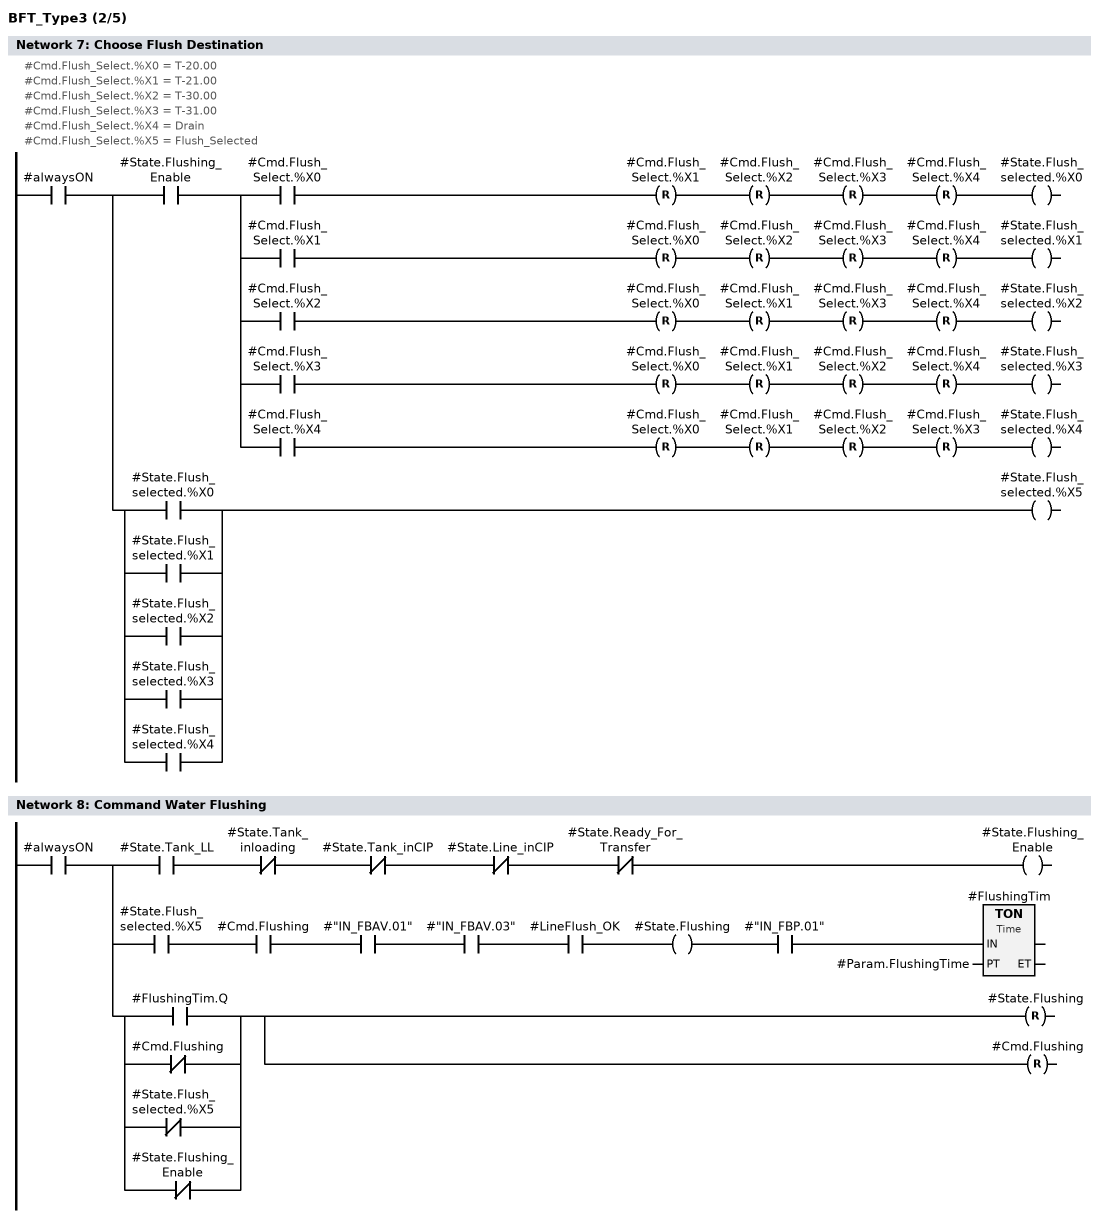
   RUNG wire#powerrail
      Contact( #alwaysON )
      wire#w1
      Contact( #State.Flushing_Enable )
      wire#w2
      Contact( #Cmd.Flush_Select.%X0 )
      R_Coil( #Cmd.Flush_Select.%X1 )
      R_Coil( #Cmd.Flush_Select.%X2 )
      R_Coil( #Cmd.Flush_Select.%X3 )
      R_Coil( #Cmd.Flush_Select.%X4 )
      Coil( #State.Flush_selected.%X0 )
   END_RUNG
   RUNG wire#w2
      Contact( #Cmd.Flush_Select.%X1 )
      R_Coil( #Cmd.Flush_Select.%X0 )
      R_Coil( #Cmd.Flush_Select.%X2 )
      R_Coil( #Cmd.Flush_Select.%X3 )
      R_Coil( #Cmd.Flush_Select.%X4 )
      Coil( #State.Flush_selected.%X1 )
   END_RUNG
   RUNG wire#w2
      Contact( #Cmd.Flush_Select.%X2 )
      R_Coil( #Cmd.Flush_Select.%X0 )
      R_Coil( #Cmd.Flush_Select.%X1 )
      R_Coil( #Cmd.Flush_Select.%X3 )
      R_Coil( #Cmd.Flush_Select.%X4 )
      Coil( #State.Flush_selected.%X2 )
   END_RUNG
   RUNG wire#w2
      Contact( #Cmd.Flush_Select.%X3 )
      R_Coil( #Cmd.Flush_Select.%X0 )
      R_Coil( #Cmd.Flush_Select.%X1 )
      R_Coil( #Cmd.Flush_Select.%X2 )
      R_Coil( #Cmd.Flush_Select.%X4 )
      Coil( #State.Flush_selected.%X3 )
   END_RUNG
   RUNG wire#w2
      Contact( #Cmd.Flush_Select.%X4 )
      R_Coil( #Cmd.Flush_Select.%X0 )
      R_Coil( #Cmd.Flush_Select.%X1 )
      R_Coil( #Cmd.Flush_Select.%X2 )
      R_Coil( #Cmd.Flush_Select.%X3 )
      Coil( #State.Flush_selected.%X4 )
   END_RUNG
   RUNG wire#w1
      Contact( #State.Flush_selected.%X0 )
      wire#w3
      Coil( #State.Flush_selected.%X5 )
   END_RUNG
   RUNG wire#w1
      Contact( #State.Flush_selected.%X1 )
   END_RUNG wire#w3
   RUNG wire#w1
      Contact( #State.Flush_selected.%X2 )
   END_RUNG wire#w3
   RUNG wire#w1
      Contact( #State.Flush_selected.%X3 )
   END_RUNG wire#w3
   RUNG wire#w1
      Contact( #State.Flush_selected.%X4 )
   END_RUNG wire#w3
   // the same network as SCL:
   #_w1 := #alwaysON AND #State.Flushing_Enable;
   #_w2 := #_w1 AND #Cmd.Flush_Select.%X0;
   IF #_w2 THEN
       #Cmd.Flush_Select.%X1 := FALSE;
       #Cmd.Flush_Select.%X2 := FALSE;
       #Cmd.Flush_Select.%X3 := FALSE;
       #Cmd.Flush_Select.%X4 := FALSE;
   END_IF;
   #State.Flush_selected.%X0 := #_w2;
   #_w3 := #_w1 AND #Cmd.Flush_Select.%X1;
   IF #_w3 THEN
       #Cmd.Flush_Select.%X0 := FALSE;
       #Cmd.Flush_Select.%X2 := FALSE;
       #Cmd.Flush_Select.%X3 := FALSE;
       #Cmd.Flush_Select.%X4 := FALSE;
   END_IF;
   #State.Flush_selected.%X1 := #_w3;
   #_w4 := #_w1 AND #Cmd.Flush_Select.%X2;
   IF #_w4 THEN
       #Cmd.Flush_Select.%X0 := FALSE;
       #Cmd.Flush_Select.%X1 := FALSE;
       #Cmd.Flush_Select.%X3 := FALSE;
       #Cmd.Flush_Select.%X4 := FALSE;
   END_IF;
   #State.Flush_selected.%X2 := #_w4;
   #_w5 := #_w1 AND #Cmd.Flush_Select.%X3;
   IF #_w5 THEN
       #Cmd.Flush_Select.%X0 := FALSE;
       #Cmd.Flush_Select.%X1 := FALSE;
       #Cmd.Flush_Select.%X2 := FALSE;
       #Cmd.Flush_Select.%X4 := FALSE;
   END_IF;
   #State.Flush_selected.%X3 := #_w5;
   #_w6 := #_w1 AND #Cmd.Flush_Select.%X4;
   IF #_w6 THEN
       #Cmd.Flush_Select.%X0 := FALSE;
       #Cmd.Flush_Select.%X1 := FALSE;
       #Cmd.Flush_Select.%X2 := FALSE;
       #Cmd.Flush_Select.%X3 := FALSE;
   END_IF;
   #State.Flush_selected.%X4 := #_w6;
   #State.Flush_selected.%X5 := #alwaysON AND (#State.Flush_selected.%X0 OR #State.Flush_selected.%X1 OR #State.Flush_selected.%X2 OR #State.Flush_selected.%X3 OR #State.Flush_selected.%X4);
END_REGION

REGION Network 8: Command Water Flushing
   RUNG wire#powerrail
      Contact( #alwaysON )
      wire#w1
      Contact( #State.Tank_LL )
      I_Contact( #State.Tank_inloading )
      I_Contact( #State.Tank_inCIP )
      I_Contact( #State.Line_inCIP )
      I_Contact( #State.Ready_For_Transfer )
      Coil( #State.Flushing_Enable )
   END_RUNG
   RUNG wire#w1
      Contact( #State.Flush_selected.%X5 )
      Contact( #Cmd.Flushing )
      Contact( #"IN_FBAV.01" )
      Contact( #"IN_FBAV.03" )
      Contact( #LineFlush_OK )
      Coil( #State.Flushing )
      Contact( #"IN_FBP.01" )
      { S7_Templates := "time_type := Time" } #FlushingTim.TON(pt := #Param.FlushingTime, et =>)
   END_RUNG
   RUNG wire#w1
      Contact( #FlushingTim.Q )
      wire#w2
      R_Coil( #State.Flushing )
   END_RUNG
   RUNG wire#w1
      I_Contact( #Cmd.Flushing )
   END_RUNG wire#w2
   RUNG wire#w1
      I_Contact( #State.Flush_selected.%X5 )
   END_RUNG wire#w2
   RUNG wire#w1
      I_Contact( #State.Flushing_Enable )
   END_RUNG wire#w2
   RUNG wire#w2
      R_Coil( #Cmd.Flushing )
   END_RUNG
   // the same network as SCL:
   #State.Flushing_Enable := #alwaysON AND #State.Tank_LL AND NOT #State.Tank_inloading AND NOT #State.Tank_inCIP AND NOT #State.Line_inCIP AND NOT #State.Ready_For_Transfer;
   #State.Flushing := #alwaysON AND #State.Flush_selected.%X5 AND #Cmd.Flushing AND #"IN_FBAV.01" AND #"IN_FBAV.03" AND #LineFlush_OK;
   #FlushingTim(IN := #State.Flushing AND #"IN_FBP.01", PT := #Param.FlushingTime);   // TON
   IF #alwaysON AND (#FlushingTim.Q OR NOT #Cmd.Flushing OR NOT #State.Flush_selected.%X5 OR NOT #State.Flushing_Enable) THEN
       #State.Flushing := FALSE;
       #Cmd.Flushing := FALSE;
   END_IF;
END_REGION

REGION Network 9: Flushing Destination AV and Pump
   // #Cmd.Flush_Select.%X0 = T-20.00
   // #Cmd.Flush_Select.%X1 = T-21.00
   // #Cmd.Flush_Select.%X2 = T-30.00
   // #Cmd.Flush_Select.%X3 = T-31.00
   // #Cmd.Flush_Select.%X4 = Drain
   // #Cmd.Flush_Select.%X5 = Flush_Selected
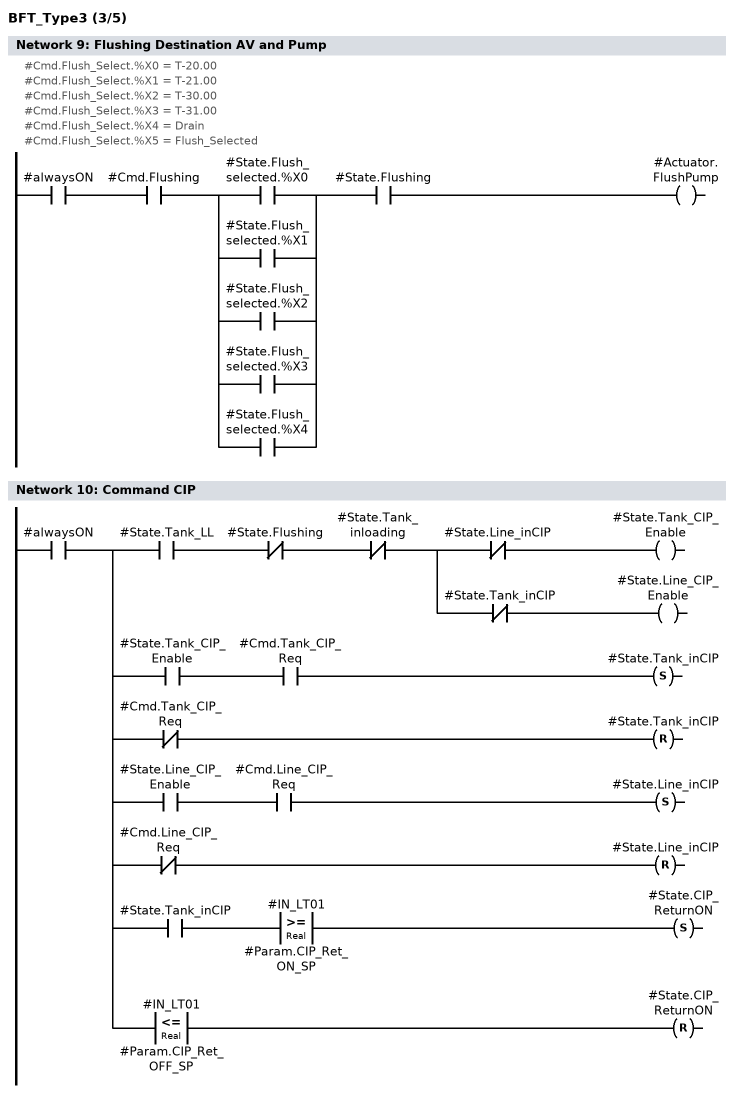
   RUNG wire#powerrail
      Contact( #alwaysON )
      Contact( #Cmd.Flushing )
      wire#w1
      Contact( #State.Flush_selected.%X0 )
      wire#w2
      Contact( #State.Flushing )
      Coil( #Actuator.FlushPump )
   END_RUNG
   RUNG wire#w1
      Contact( #State.Flush_selected.%X1 )
   END_RUNG wire#w2
   RUNG wire#w1
      Contact( #State.Flush_selected.%X2 )
   END_RUNG wire#w2
   RUNG wire#w1
      Contact( #State.Flush_selected.%X3 )
   END_RUNG wire#w2
   RUNG wire#w1
      Contact( #State.Flush_selected.%X4 )
   END_RUNG wire#w2
   // the same network as SCL:
   #Actuator.FlushPump := #alwaysON AND #Cmd.Flushing AND (#State.Flush_selected.%X0 OR #State.Flush_selected.%X1 OR #State.Flush_selected.%X2 OR #State.Flush_selected.%X3 OR #State.Flush_selected.%X4) AND #State.Flushing;
END_REGION

REGION Network 10: Command CIP
   RUNG wire#powerrail
      Contact( #alwaysON )
      wire#w1
      Contact( #State.Tank_LL )
      I_Contact( #State.Flushing )
      I_Contact( #State.Tank_inloading )
      wire#w2
      I_Contact( #State.Line_inCIP )
      Coil( #State.Tank_CIP_Enable )
   END_RUNG
   RUNG wire#w2
      I_Contact( #State.Tank_inCIP )
      Coil( #State.Line_CIP_Enable )
   END_RUNG
   RUNG wire#w1
      Contact( #State.Tank_CIP_Enable )
      Contact( #Cmd.Tank_CIP_Req )
      S_Coil( #State.Tank_inCIP )
   END_RUNG
   RUNG wire#w1
      I_Contact( #Cmd.Tank_CIP_Req )
      R_Coil( #State.Tank_inCIP )
   END_RUNG
   RUNG wire#w1
      Contact( #State.Line_CIP_Enable )
      Contact( #Cmd.Line_CIP_Req )
      S_Coil( #State.Line_inCIP )
   END_RUNG
   RUNG wire#w1
      I_Contact( #Cmd.Line_CIP_Req )
      R_Coil( #State.Line_inCIP )
   END_RUNG
   RUNG wire#w1
      Contact( #State.Tank_inCIP )
      { S7_Templates := "SrcType := Real" } GE_Contact(in1 := #IN_LT01, in2 := #Param.CIP_Ret_ON_SP)
      S_Coil( #State.CIP_ReturnON )
   END_RUNG
   RUNG wire#w1
      { S7_Templates := "SrcType := Real" } LE_Contact(in1 := #IN_LT01, in2 := #Param.CIP_Ret_OFF_SP)
      R_Coil( #State.CIP_ReturnON )
   END_RUNG
   // the same network as SCL:
   #_w1 := #alwaysON AND #State.Tank_LL AND NOT #State.Flushing AND NOT #State.Tank_inloading;
   #State.Tank_CIP_Enable := #_w1 AND NOT #State.Line_inCIP;
   #State.Line_CIP_Enable := #_w1 AND NOT #State.Tank_inCIP;
   IF #alwaysON AND #State.Tank_CIP_Enable AND #Cmd.Tank_CIP_Req THEN #State.Tank_inCIP := TRUE; END_IF;
   IF #alwaysON AND NOT #Cmd.Tank_CIP_Req THEN #State.Tank_inCIP := FALSE; END_IF;
   IF #alwaysON AND #State.Line_CIP_Enable AND #Cmd.Line_CIP_Req THEN #State.Line_inCIP := TRUE; END_IF;
   IF #alwaysON AND NOT #Cmd.Line_CIP_Req THEN #State.Line_inCIP := FALSE; END_IF;
   IF #alwaysON AND #State.Tank_inCIP AND (#IN_LT01 >= #Param.CIP_Ret_ON_SP) THEN
       #State.CIP_ReturnON := TRUE;
   END_IF;
   IF #alwaysON AND (#IN_LT01 <= #Param.CIP_Ret_OFF_SP) THEN #State.CIP_ReturnON := FALSE; END_IF;
END_REGION

REGION Network 11: Loading AV and Pump
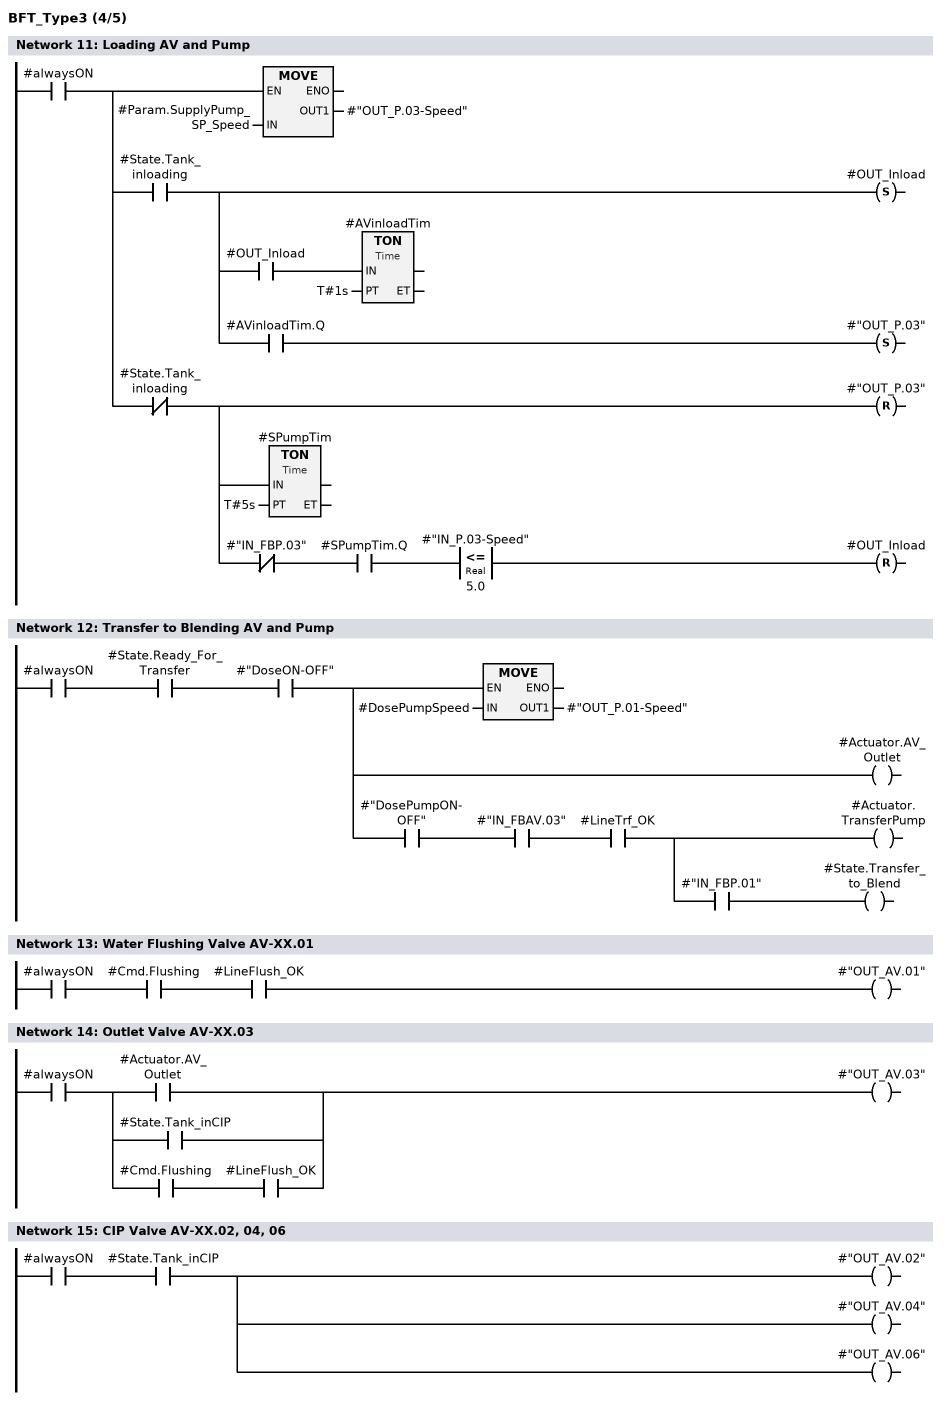
   RUNG wire#powerrail
      Contact( #alwaysON )
      wire#w1
      Move(in := #Param.SupplyPump_SP_Speed, out1 => #"OUT_P.03-Speed")
   END_RUNG
   RUNG wire#w1
      Contact( #State.Tank_inloading )
      wire#w2
      S_Coil( #OUT_Inload )
   END_RUNG
   RUNG wire#w2
      Contact( #OUT_Inload )
      { S7_Templates := "time_type := Time" } #AVinloadTim.TON(pt := T#1s, et =>)
   END_RUNG
   RUNG wire#w2
      Contact( #AVinloadTim.Q )
      S_Coil( #"OUT_P.03" )
   END_RUNG
   RUNG wire#w1
      I_Contact( #State.Tank_inloading )
      wire#w3
      R_Coil( #"OUT_P.03" )
   END_RUNG
   RUNG wire#w3
      { S7_Templates := "time_type := Time" } #SPumpTim.TON(pt := T#5s, et =>)
   END_RUNG
   RUNG wire#w3
      I_Contact( #"IN_FBP.03" )
      Contact( #SPumpTim.Q )
      { S7_Templates := "SrcType := Real" } LE_Contact(in1 := #"IN_P.03-Speed", in2 := 5.0)
      R_Coil( #OUT_Inload )
   END_RUNG
   // the same network as SCL:
   IF #alwaysON THEN #"OUT_P.03-Speed" := #Param.SupplyPump_SP_Speed; END_IF;
   #_w1 := #alwaysON AND #State.Tank_inloading;
   IF #_w1 THEN #OUT_Inload := TRUE; END_IF;
   #AVinloadTim(IN := #_w1 AND #OUT_Inload, PT := T#1s);   // TON
   IF #_w1 AND #AVinloadTim.Q THEN #"OUT_P.03" := TRUE; END_IF;
   #_w2 := #alwaysON AND NOT #State.Tank_inloading;
   IF #_w2 THEN #"OUT_P.03" := FALSE; END_IF;
   #SPumpTim(IN := #_w2, PT := T#5s);   // TON
   IF #_w2 AND NOT #"IN_FBP.03" AND #SPumpTim.Q AND (#"IN_P.03-Speed" <= 5.0) THEN
       #OUT_Inload := FALSE;
   END_IF;
END_REGION

REGION Network 12: Transfer to Blending AV and Pump
   RUNG wire#powerrail
      Contact( #alwaysON )
      Contact( #State.Ready_For_Transfer )
      Contact( #"DoseON-OFF" )
      wire#w1
      Move(in := #DosePumpSpeed, out1 => #"OUT_P.01-Speed")
   END_RUNG
   RUNG wire#w1
      Coil( #Actuator.AV_Outlet )
   END_RUNG
   RUNG wire#w1
      Contact( #"DosePumpON-OFF" )
      Contact( #"IN_FBAV.03" )
      Contact( #LineTrf_OK )
      wire#w2
      Coil( #Actuator.TransferPump )
   END_RUNG
   RUNG wire#w2
      Contact( #"IN_FBP.01" )
      Coil( #State.Transfer_to_Blend )
   END_RUNG
   // the same network as SCL:
   #_w1 := #alwaysON AND #State.Ready_For_Transfer AND #"DoseON-OFF";
   IF #_w1 THEN #"OUT_P.01-Speed" := #DosePumpSpeed; END_IF;
   #Actuator.AV_Outlet := #_w1;
   #Actuator.TransferPump := #_w1 AND #"DosePumpON-OFF" AND #"IN_FBAV.03" AND #LineTrf_OK;
   #State.Transfer_to_Blend := #Actuator.TransferPump AND #"IN_FBP.01";
END_REGION

REGION Network 13: Water Flushing Valve AV-XX.01
   RUNG wire#powerrail
      Contact( #alwaysON )
      Contact( #Cmd.Flushing )
      Contact( #LineFlush_OK )
      Coil( #"OUT_AV.01" )
   END_RUNG
   // the same network as SCL:
   #"OUT_AV.01" := #alwaysON AND #Cmd.Flushing AND #LineFlush_OK;
END_REGION

REGION Network 14: Outlet Valve AV-XX.03
   RUNG wire#powerrail
      Contact( #alwaysON )
      wire#w1
      Contact( #Actuator.AV_Outlet )
      wire#w2
      Coil( #"OUT_AV.03" )
   END_RUNG
   RUNG wire#w1
      Contact( #State.Tank_inCIP )
   END_RUNG wire#w2
   RUNG wire#w1
      Contact( #Cmd.Flushing )
      Contact( #LineFlush_OK )
   END_RUNG wire#w2
   // the same network as SCL:
   #"OUT_AV.03" := #alwaysON AND (#Actuator.AV_Outlet OR #State.Tank_inCIP OR (#Cmd.Flushing AND #LineFlush_OK));
END_REGION

REGION Network 15: CIP Valve AV-XX.02, 04, 06
   RUNG wire#powerrail
      Contact( #alwaysON )
      Contact( #State.Tank_inCIP )
      wire#w1
      Coil( #"OUT_AV.02" )
   END_RUNG
   RUNG wire#w1
      Coil( #"OUT_AV.04" )
   END_RUNG
   RUNG wire#w1
      Coil( #"OUT_AV.06" )
   END_RUNG
   // the same network as SCL:
   #"OUT_AV.02" := #alwaysON AND #State.Tank_inCIP;
   #"OUT_AV.04" := #"OUT_AV.02";
   #"OUT_AV.06" := #"OUT_AV.02";
END_REGION

REGION Network 16: Line CIP Valve AV-XX.05,12
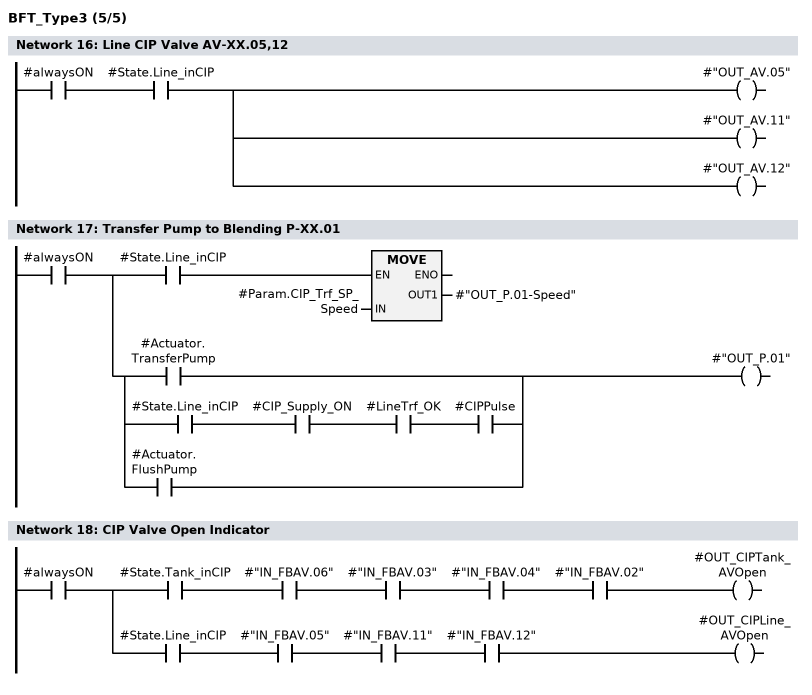
   RUNG wire#powerrail
      Contact( #alwaysON )
      Contact( #State.Line_inCIP )
      wire#w1
      Coil( #"OUT_AV.05" )
   END_RUNG
   RUNG wire#w1
      Coil( #"OUT_AV.11" )
   END_RUNG
   RUNG wire#w1
      Coil( #"OUT_AV.12" )
   END_RUNG
   // the same network as SCL:
   #"OUT_AV.05" := #alwaysON AND #State.Line_inCIP;
   #"OUT_AV.11" := #"OUT_AV.05";
   #"OUT_AV.12" := #"OUT_AV.05";
END_REGION

REGION Network 17: Transfer Pump to Blending P-XX.01
   RUNG wire#powerrail
      Contact( #alwaysON )
      wire#w1
      Contact( #State.Line_inCIP )
      Move(in := #Param.CIP_Trf_SP_Speed, out1 => #"OUT_P.01-Speed")
   END_RUNG
   RUNG wire#w1
      Contact( #Actuator.TransferPump )
      wire#w2
      Coil( #"OUT_P.01" )
   END_RUNG
   RUNG wire#w1
      Contact( #State.Line_inCIP )
      Contact( #CIP_Supply_ON )
      Contact( #LineTrf_OK )
      Contact( #CIPPulse )
   END_RUNG wire#w2
   RUNG wire#w1
      Contact( #Actuator.FlushPump )
   END_RUNG wire#w2
   // the same network as SCL:
   IF #alwaysON AND #State.Line_inCIP THEN #"OUT_P.01-Speed" := #Param.CIP_Trf_SP_Speed; END_IF;
   #"OUT_P.01" := #alwaysON AND (#Actuator.TransferPump OR (#State.Line_inCIP AND #CIP_Supply_ON AND #LineTrf_OK AND #CIPPulse) OR #Actuator.FlushPump);
END_REGION

REGION Network 18: CIP Valve Open Indicator
   RUNG wire#powerrail
      Contact( #alwaysON )
      wire#w1
      Contact( #State.Tank_inCIP )
      Contact( #"IN_FBAV.06" )
      Contact( #"IN_FBAV.03" )
      Contact( #"IN_FBAV.04" )
      Contact( #"IN_FBAV.02" )
      Coil( #OUT_CIPTank_AVOpen )
   END_RUNG
   RUNG wire#w1
      Contact( #State.Line_inCIP )
      Contact( #"IN_FBAV.05" )
      Contact( #"IN_FBAV.11" )
      Contact( #"IN_FBAV.12" )
      Coil( #OUT_CIPLine_AVOpen )
   END_RUNG
   // the same network as SCL:
   #OUT_CIPTank_AVOpen := #alwaysON AND #State.Tank_inCIP AND #"IN_FBAV.06" AND #"IN_FBAV.03" AND #"IN_FBAV.04" AND #"IN_FBAV.02";
   #OUT_CIPLine_AVOpen := #alwaysON AND #State.Line_inCIP AND #"IN_FBAV.05" AND #"IN_FBAV.11" AND #"IN_FBAV.12";
END_REGION
END_FUNCTION_BLOCK

DATA_BLOCK "Alarm_Collector_Gen_DB"   // DB65
VERSION : 0.1
// stored: AutoNumber true, DBAccessibleFromOPCUA true, DBAccessibleFromWebserver true, InstanceOfName Alarm_Collector_Gen, InstanceOfType FB
"Alarm_Collector_Gen"
BEGIN
END_DATA_BLOCK

DATA_BLOCK "ReadDateandTime_DB"   // DB31
VERSION : 0.1
// stored: AutoNumber false, DBAccessibleFromOPCUA true, DBAccessibleFromWebserver true, InstanceOfName ReadDateandTime, InstanceOfType FB
"ReadDateandTime"
BEGIN
END_DATA_BLOCK

DATA_BLOCK "Sim_PTM_DB"   // DB1000
VERSION : 0.1
// stored: AutoNumber false, DBAccessibleFromOPCUA true, DBAccessibleFromWebserver true, InstanceOfName Sim_PT1, InstanceOfType FB
"Sim_PT1"
   // VAR_INPUT
   //    Reset : Bool;
   //    Calc_Param : Bool;
   //    Input : Real;
   //    TM_LAG1 : Real;
   //    GAIN : Real;
   //    Cycle : Real;
   //    Max_Out : Real;
   //    AMB_TEM : Real;
   // END_VAR
   // VAR_OUTPUT
   //    Max_reached : Bool;
   //    Output : Real;
   // END_VAR
   // VAR
   //    r_f1 : Real;
   //    r_e1 : Real;
   //    overfirst : Bool;
   // END_VAR
BEGIN
END_DATA_BLOCK

DATA_BLOCK "Sim_PTS_DB"   // DB1001
VERSION : 0.1
// stored: AutoNumber false, DBAccessibleFromOPCUA true, DBAccessibleFromWebserver true, InstanceOfName Sim_PT1, InstanceOfType FB
"Sim_PT1"
   // VAR_INPUT
   //    Reset : Bool;
   //    Calc_Param : Bool;
   //    Input : Real;
   //    TM_LAG1 : Real;
   //    GAIN : Real;
   //    Cycle : Real;
   //    Max_Out : Real;
   //    AMB_TEM : Real;
   // END_VAR
   // VAR_OUTPUT
   //    Max_reached : Bool;
   //    Output : Real;
   // END_VAR
   // VAR
   //    r_f1 : Real;
   //    r_e1 : Real;
   //    overfirst : Bool;
   // END_VAR
BEGIN
END_DATA_BLOCK

DATA_BLOCK "AlarmFlowColletor"   // DB217
VERSION : 0.1
// stored: AutoNumber false, DBAccessibleFromOPCUA true, DBAccessibleFromWebserver true, InstanceOfName Alarm Flow Collector, InstanceOfType FB
"Alarm Flow Collector"
BEGIN
END_DATA_BLOCK

DATA_BLOCK "Blend_T-20"   // DB211
VERSION : 0.1
// stored: AutoNumber false, DBAccessibleFromOPCUA true, DBAccessibleFromWebserver true, InstanceOfName Blend_Tank, InstanceOfType FB
"Blend_Tank"
BEGIN
END_DATA_BLOCK

DATA_BLOCK "Blend_T-21"   // DB212
VERSION : 0.1
// stored: AutoNumber false, DBAccessibleFromOPCUA true, DBAccessibleFromWebserver true, InstanceOfName Blend_Tank, InstanceOfType FB
"Blend_Tank"
BEGIN
END_DATA_BLOCK

DATA_BLOCK "Blend_T-30"   // DB213
VERSION : 0.1
// stored: AutoNumber false, DBAccessibleFromOPCUA true, DBAccessibleFromWebserver true, InstanceOfName Blend_Tank, InstanceOfType FB
"Blend_Tank"
BEGIN
END_DATA_BLOCK

DATA_BLOCK "Blend_T-31"   // DB214
VERSION : 0.1
// stored: AutoNumber false, DBAccessibleFromOPCUA true, DBAccessibleFromWebserver true, InstanceOfName Blend_Tank, InstanceOfType FB
"Blend_Tank"
BEGIN
END_DATA_BLOCK

DATA_BLOCK "Blend_T-40"   // DB215
VERSION : 0.1
// stored: AutoNumber false, DBAccessibleFromOPCUA true, DBAccessibleFromWebserver true, InstanceOfName Blend_Tank, InstanceOfType FB
"Blend_Tank"
BEGIN
END_DATA_BLOCK

DATA_BLOCK "Blend_T-41"   // DB216
VERSION : 0.1
// stored: AutoNumber false, DBAccessibleFromOPCUA true, DBAccessibleFromWebserver true, InstanceOfName Blend_Tank, InstanceOfType FB
"Blend_Tank"
BEGIN
END_DATA_BLOCK

DATA_BLOCK "GetData_DB"   // DB45
AUTHOR : SiemensIndustryOnlineSupport
FAMILY : S7comm
VERSION : 1.0
// stored: AutoNumber true, DBAccessibleFromOPCUA true, DBAccessibleFromWebserver true, InstanceOfName GetData, InstanceOfType FB
"GetData"
   // VAR_INPUT
   //    execute : Bool;
   //    connectionId : Word;
   // END_VAR
   // VAR_OUTPUT
   //    done { ExternalWritable := 'False'} : Bool;
   //    busy { ExternalWritable := 'False'} : Bool;
   //    error { ExternalWritable := 'False'} : Bool;
   //    status { ExternalWritable := 'False'} : Word;
   // END_VAR
   // VAR_IN_OUT
   //    ADDR_1 : Remote;
   //    ADDR_2 : Remote;
   //    ADDR_3 : Remote;
   //    ADDR_4 : Remote;
   //    RD_1 : Variant;
   //    RD_2 : Variant;
   //    RD_3 : Variant;
   //    RD_4 : Variant;
   // END_VAR
   // VAR
   //    statExecuteOld { ExternalAccessible := 'False'; ExternalVisible := 'False'; ExternalWritable := 'False'} : Bool;
   //    statDone { ExternalAccessible := 'False'; ExternalVisible := 'False'; ExternalWritable := 'False'} : Bool;
   //    statBusy { ExternalAccessible := 'False'; ExternalVisible := 'False'; ExternalWritable := 'False'} : Bool;
   //    statError { ExternalAccessible := 'False'; ExternalVisible := 'False'; ExternalWritable := 'False'} : Bool;
   //    statStatus { ExternalAccessible := 'False'; ExternalVisible := 'False'; ExternalWritable := 'False'} : Word;
   //    statFBState { ExternalAccessible := 'False'; ExternalVisible := 'False'; ExternalWritable := 'False'} : DInt;
   //    instGet { S7_SetPoint := 'True'} : GET;
   //    statErrorGet { S7_SetPoint := 'True'} : Bool;
   // END_VAR
BEGIN
END_DATA_BLOCK

DATA_BLOCK "THE1_GetData_DB"   // DB16
AUTHOR : SiemensIndustryOnlineSupport
FAMILY : S7comm
VERSION : 1.0
// stored: AutoNumber true, DBAccessibleFromOPCUA true, DBAccessibleFromWebserver true, InstanceOfName GetData, InstanceOfType FB
"GetData"
   // VAR_INPUT
   //    execute : Bool;
   //    connectionId : Word;
   // END_VAR
   // VAR_OUTPUT
   //    done { ExternalWritable := 'False'} : Bool;
   //    busy { ExternalWritable := 'False'} : Bool;
   //    error { ExternalWritable := 'False'} : Bool;
   //    status { ExternalWritable := 'False'} : Word;
   // END_VAR
   // VAR_IN_OUT
   //    ADDR_1 : Remote;
   //    ADDR_2 : Remote;
   //    ADDR_3 : Remote;
   //    ADDR_4 : Remote;
   //    RD_1 : Variant;
   //    RD_2 : Variant;
   //    RD_3 : Variant;
   //    RD_4 : Variant;
   // END_VAR
   // VAR
   //    statExecuteOld { ExternalAccessible := 'False'; ExternalVisible := 'False'; ExternalWritable := 'False'} : Bool;
   //    statDone { ExternalAccessible := 'False'; ExternalVisible := 'False'; ExternalWritable := 'False'} : Bool;
   //    statBusy { ExternalAccessible := 'False'; ExternalVisible := 'False'; ExternalWritable := 'False'} : Bool;
   //    statError { ExternalAccessible := 'False'; ExternalVisible := 'False'; ExternalWritable := 'False'} : Bool;
   //    statStatus { ExternalAccessible := 'False'; ExternalVisible := 'False'; ExternalWritable := 'False'} : Word;
   //    statFBState { ExternalAccessible := 'False'; ExternalVisible := 'False'; ExternalWritable := 'False'} : DInt;
   //    instGet { S7_SetPoint := 'True'} : GET;
   //    statErrorGet { S7_SetPoint := 'True'} : Bool;
   // END_VAR
BEGIN
END_DATA_BLOCK

DATA_BLOCK "THE2_GetData_DB"   // DB17
AUTHOR : SiemensIndustryOnlineSupport
FAMILY : S7comm
VERSION : 1.0
// stored: AutoNumber true, DBAccessibleFromOPCUA true, DBAccessibleFromWebserver true, InstanceOfName GetData, InstanceOfType FB
"GetData"
   // VAR_INPUT
   //    execute : Bool;
   //    connectionId : Word;
   // END_VAR
   // VAR_OUTPUT
   //    done { ExternalWritable := 'False'} : Bool;
   //    busy { ExternalWritable := 'False'} : Bool;
   //    error { ExternalWritable := 'False'} : Bool;
   //    status { ExternalWritable := 'False'} : Word;
   // END_VAR
   // VAR_IN_OUT
   //    ADDR_1 : Remote;
   //    ADDR_2 : Remote;
   //    ADDR_3 : Remote;
   //    ADDR_4 : Remote;
   //    RD_1 : Variant;
   //    RD_2 : Variant;
   //    RD_3 : Variant;
   //    RD_4 : Variant;
   // END_VAR
   // VAR
   //    statExecuteOld { ExternalAccessible := 'False'; ExternalVisible := 'False'; ExternalWritable := 'False'} : Bool;
   //    statDone { ExternalAccessible := 'False'; ExternalVisible := 'False'; ExternalWritable := 'False'} : Bool;
   //    statBusy { ExternalAccessible := 'False'; ExternalVisible := 'False'; ExternalWritable := 'False'} : Bool;
   //    statError { ExternalAccessible := 'False'; ExternalVisible := 'False'; ExternalWritable := 'False'} : Bool;
   //    statStatus { ExternalAccessible := 'False'; ExternalVisible := 'False'; ExternalWritable := 'False'} : Word;
   //    statFBState { ExternalAccessible := 'False'; ExternalVisible := 'False'; ExternalWritable := 'False'} : DInt;
   //    instGet { S7_SetPoint := 'True'} : GET;
   //    statErrorGet { S7_SetPoint := 'True'} : Bool;
   // END_VAR
BEGIN
END_DATA_BLOCK

DATA_BLOCK "T-12.00_Homomixer"   // DB102
VERSION : 0.1
// stored: AutoNumber false, DBAccessibleFromOPCUA true, DBAccessibleFromWebserver true, InstanceOfName Homomix, InstanceOfType FB
"Homomix"
BEGIN
END_DATA_BLOCK

DATA_BLOCK "T-13.00_Homomixer"   // DB103
VERSION : 0.1
// stored: AutoNumber false, DBAccessibleFromOPCUA true, DBAccessibleFromWebserver true, InstanceOfName Homomix, InstanceOfType FB
"Homomix"
BEGIN
END_DATA_BLOCK

DATA_BLOCK "T-14.00_Homomixer"   // DB104
VERSION : 0.1
// stored: AutoNumber false, DBAccessibleFromOPCUA true, DBAccessibleFromWebserver true, InstanceOfName Homomix, InstanceOfType FB
"Homomix"
BEGIN
END_DATA_BLOCK

DATA_BLOCK "T-23.00"   // DB37
VERSION : 0.1
// stored: AutoNumber false, DBAccessibleFromOPCUA true, DBAccessibleFromWebserver true, InstanceOfName Storage_Tank_Multi_Inload, InstanceOfType FB
"Storage_Tank_Multi_Inload"
BEGIN
END_DATA_BLOCK

DATA_BLOCK "T-24.00"   // DB55
VERSION : 0.1
// stored: AutoNumber false, DBAccessibleFromOPCUA true, DBAccessibleFromWebserver true, InstanceOfName Storage_Tank_Multi_Inload, InstanceOfType FB
"Storage_Tank_Multi_Inload"
BEGIN
END_DATA_BLOCK

DATA_BLOCK "T-29.00"   // DB38
VERSION : 0.1
// stored: AutoNumber true, DBAccessibleFromOPCUA true, DBAccessibleFromWebserver true, InstanceOfName Storage_Tank_Single_Inload, InstanceOfType FB
"Storage_Tank_Single_Inload"
BEGIN
END_DATA_BLOCK

DATA_BLOCK "T-33.00"   // DB41
VERSION : 0.1
// stored: AutoNumber false, DBAccessibleFromOPCUA true, DBAccessibleFromWebserver true, InstanceOfName Storage_Tank_Multi_Inload, InstanceOfType FB
"Storage_Tank_Multi_Inload"
BEGIN
END_DATA_BLOCK

DATA_BLOCK "T-34.00"   // DB42
VERSION : 0.1
// stored: AutoNumber false, DBAccessibleFromOPCUA true, DBAccessibleFromWebserver true, InstanceOfName Storage_Tank_Multi_Inload, InstanceOfType FB
"Storage_Tank_Multi_Inload"
BEGIN
END_DATA_BLOCK

DATA_BLOCK "T-35.00"   // DB43
VERSION : 0.1
// stored: AutoNumber false, DBAccessibleFromOPCUA true, DBAccessibleFromWebserver true, InstanceOfName Storage_Tank_Multi_Inload, InstanceOfType FB
"Storage_Tank_Multi_Inload"
BEGIN
END_DATA_BLOCK

DATA_BLOCK "T-39.00"   // DB40
VERSION : 0.1
// stored: AutoNumber false, DBAccessibleFromOPCUA true, DBAccessibleFromWebserver true, InstanceOfName Storage_Tank_Single_Inload, InstanceOfType FB
"Storage_Tank_Single_Inload"
BEGIN
END_DATA_BLOCK

DATA_BLOCK "T-79.00"   // DB54
VERSION : 0.1
// stored: AutoNumber false, DBAccessibleFromOPCUA true, DBAccessibleFromWebserver true, InstanceOfName Storage_Tank_Multi_Inload, InstanceOfType FB
"Storage_Tank_Multi_Inload"
BEGIN
END_DATA_BLOCK

DATA_BLOCK "T-81.00"   // DB51
VERSION : 0.1
// stored: AutoNumber false, DBAccessibleFromOPCUA true, DBAccessibleFromWebserver true, InstanceOfName Storage_Tank_Multi_Inload, InstanceOfType FB
"Storage_Tank_Multi_Inload"
BEGIN
END_DATA_BLOCK

DATA_BLOCK "T-84.00"   // DB53
VERSION : 0.1
// stored: AutoNumber false, DBAccessibleFromOPCUA true, DBAccessibleFromWebserver true, InstanceOfName Storage_Tank_Multi_Inload, InstanceOfType FB
"Storage_Tank_Multi_Inload"
BEGIN
END_DATA_BLOCK

DATA_BLOCK "T-85.00"   // DB52
VERSION : 0.1
// stored: AutoNumber false, DBAccessibleFromOPCUA true, DBAccessibleFromWebserver true, InstanceOfName Storage_Tank_Multi_Inload, InstanceOfType FB
"Storage_Tank_Multi_Inload"
BEGIN
END_DATA_BLOCK

DATA_BLOCK "T-02_ChiliAwetan_1"   // DB361
VERSION : 0.1
// stored: AutoNumber false, DBAccessibleFromOPCUA true, DBAccessibleFromWebserver true, InstanceOfName BFT_ChiliAwetan, InstanceOfType FB
"BFT_ChiliAwetan"
BEGIN
END_DATA_BLOCK

DATA_BLOCK "T-03_ChiliAwetan_2"   // DB362
VERSION : 0.1
// stored: AutoNumber false, DBAccessibleFromOPCUA true, DBAccessibleFromWebserver true, InstanceOfName BFT_ChiliAwetan, InstanceOfType FB
"BFT_ChiliAwetan"
BEGIN
END_DATA_BLOCK

DATA_BLOCK "T-04_ChiliAwetan_3"   // DB363
VERSION : 0.1
// stored: AutoNumber false, DBAccessibleFromOPCUA true, DBAccessibleFromWebserver true, InstanceOfName BFT_ChiliAwetan, InstanceOfType FB
"BFT_ChiliAwetan"
BEGIN
END_DATA_BLOCK

DATA_BLOCK "T-05_Tomato"   // DB364
VERSION : 0.1
// stored: AutoNumber false, DBAccessibleFromOPCUA true, DBAccessibleFromWebserver true, InstanceOfName BFT_Tomato, InstanceOfType FB
"BFT_Tomato"
BEGIN
END_DATA_BLOCK

DATA_BLOCK "T-06_ChiliFresh_1"   // DB365
VERSION : 0.1
// stored: AutoNumber false, DBAccessibleFromOPCUA true, DBAccessibleFromWebserver true, InstanceOfName BFT_ChiliFresh, InstanceOfType FB
"BFT_ChiliFresh"
BEGIN
END_DATA_BLOCK

DATA_BLOCK "T-07_ChiliFresh_2"   // DB366
VERSION : 0.1
// stored: AutoNumber false, DBAccessibleFromOPCUA true, DBAccessibleFromWebserver true, InstanceOfName BFT_ChiliFresh, InstanceOfType FB
"BFT_ChiliFresh"
BEGIN
END_DATA_BLOCK

DATA_BLOCK "T-08_ChiliFresh_3"   // DB367
VERSION : 0.1
// stored: AutoNumber false, DBAccessibleFromOPCUA true, DBAccessibleFromWebserver true, InstanceOfName BFT_ChiliFresh, InstanceOfType FB
"BFT_ChiliFresh"
BEGIN
END_DATA_BLOCK

DATA_BLOCK "T-09_Garlic"   // DB368
VERSION : 0.1
// stored: AutoNumber false, DBAccessibleFromOPCUA true, DBAccessibleFromWebserver true, InstanceOfName BFT_Garlic, InstanceOfType FB
"BFT_Garlic"
BEGIN
END_DATA_BLOCK

DATA_BLOCK "T-10_Vinegar"   // DB369
VERSION : 0.1
// stored: AutoNumber false, DBAccessibleFromOPCUA true, DBAccessibleFromWebserver true, InstanceOfName BFT_Vinegar, InstanceOfType FB
"BFT_Vinegar"
BEGIN
END_DATA_BLOCK

DATA_BLOCK "T-51_HW"   // DB370
VERSION : 0.1
// stored: AutoNumber false, DBAccessibleFromOPCUA true, DBAccessibleFromWebserver true, InstanceOfName Hot_Water, InstanceOfType FB
"Hot_Water"
BEGIN
END_DATA_BLOCK

DATA_BLOCK "BFT-61"   // DB111
VERSION : 0.1
// stored: AutoNumber false, DBAccessibleFromOPCUA true, DBAccessibleFromWebserver true, InstanceOfName Buffer_Tank, InstanceOfType FB
"Buffer_Tank"
BEGIN
END_DATA_BLOCK

DATA_BLOCK "BFT-64"   // DB112
VERSION : 0.1
// stored: AutoNumber false, DBAccessibleFromOPCUA true, DBAccessibleFromWebserver true, InstanceOfName Buffer_Tank, InstanceOfType FB
"Buffer_Tank"
BEGIN
END_DATA_BLOCK

DATA_BLOCK "BFT-65"   // DB113
VERSION : 0.1
// stored: AutoNumber false, DBAccessibleFromOPCUA true, DBAccessibleFromWebserver true, InstanceOfName Buffer_Tank, InstanceOfType FB
"Buffer_Tank"
BEGIN
END_DATA_BLOCK

DATA_BLOCK "BFT-66"   // DB114
VERSION : 0.1
// stored: AutoNumber false, DBAccessibleFromOPCUA true, DBAccessibleFromWebserver true, InstanceOfName Buffer_Tank, InstanceOfType FB
"Buffer_Tank"
BEGIN
END_DATA_BLOCK

DATA_BLOCK "BFT-67"   // DB115
VERSION : 0.1
// stored: AutoNumber false, DBAccessibleFromOPCUA true, DBAccessibleFromWebserver true, InstanceOfName Buffer_Tank, InstanceOfType FB
"Buffer_Tank"
BEGIN
END_DATA_BLOCK

DATA_BLOCK "BFT-68"   // DB116
VERSION : 0.1
// stored: AutoNumber false, DBAccessibleFromOPCUA true, DBAccessibleFromWebserver true, InstanceOfName Buffer_Tank, InstanceOfType FB
"Buffer_Tank"
BEGIN
END_DATA_BLOCK

DATA_BLOCK "Danfos_VSD_DB"   // DB46
VERSION : 0.1
// stored: AutoNumber false, DBAccessibleFromOPCUA true, DBAccessibleFromWebserver true, InstanceOfName Danfos_VSD, InstanceOfType FB
"Danfos_VSD"
BEGIN
END_DATA_BLOCK

DATA_BLOCK "IO Motor MCC Panel Blending_DB"   // DB5
VERSION : 0.1
// stored: AutoNumber true, DBAccessibleFromOPCUA true, DBAccessibleFromWebserver true, InstanceOfName IO Motor MCC Panel Blending, InstanceOfType FB
"IO Motor MCC Panel Blending"
BEGIN
   "XA-20.00".IN_SP_Speed := 5.0;
   "XA-21.00".IN_SP_Speed := 5.0;
   "P-21.01".IN_SP_Speed := 5.0;
   "XA-30.00".IN_SP_Speed := 5.0;
   "XA-31.00".IN_SP_Speed := 5.0;
   "P-31.01".IN_SP_Speed := 5.0;
   "P-32.01".IN_SP_Speed := 5.0;
   "P-32.03".IN_SP_Speed := 5.0;
END_DATA_BLOCK

DATA_BLOCK "P21.01Dan"   // DB23
VERSION : 0.1
// stored: AutoNumber true, DBAccessibleFromOPCUA true, DBAccessibleFromWebserver true, InstanceOfName Danfos_VSD, InstanceOfType FB
"Danfos_VSD"
BEGIN
END_DATA_BLOCK

DATA_BLOCK "P22.01Dan"   // DB22
VERSION : 0.1
// stored: AutoNumber true, DBAccessibleFromOPCUA true, DBAccessibleFromWebserver true, InstanceOfName Danfos_VSD, InstanceOfType FB
"Danfos_VSD"
BEGIN
END_DATA_BLOCK

DATA_BLOCK "IO Analog Homomixer_DB"   // DB2
VERSION : 0.1
// stored: AutoNumber true, DBAccessibleFromOPCUA true, DBAccessibleFromWebserver true, InstanceOfName IO Analog Homomixer, InstanceOfType FB
"IO Analog Homomixer"
BEGIN
END_DATA_BLOCK

DATA_BLOCK "IO Digital Homomixer_DB"   // DB3
VERSION : 0.1
// stored: AutoNumber true, DBAccessibleFromOPCUA true, DBAccessibleFromWebserver true, InstanceOfName IO Digital Homomixer, InstanceOfType FB
"IO Digital Homomixer"
BEGIN
END_DATA_BLOCK

DATA_BLOCK "IO Valve Homomixer_DB"   // DB4
VERSION : 0.1
// stored: AutoNumber true, DBAccessibleFromOPCUA true, DBAccessibleFromWebserver true, InstanceOfName IO Valve Homomixer, InstanceOfType FB
"IO Valve Homomixer"
BEGIN
END_DATA_BLOCK

DATA_BLOCK "IO Analog Blending_DB"   // DB6
VERSION : 0.1
// stored: AutoNumber true, DBAccessibleFromOPCUA true, DBAccessibleFromWebserver true, InstanceOfName IO Analog Blending, InstanceOfType FB
"IO Analog Blending"
BEGIN
END_DATA_BLOCK

DATA_BLOCK "IO Digital Blending_DB"   // DB7
VERSION : 0.1
// stored: AutoNumber true, DBAccessibleFromOPCUA true, DBAccessibleFromWebserver true, InstanceOfName IO Digital Blending, InstanceOfType FB
"IO Digital Blending"
BEGIN
END_DATA_BLOCK

DATA_BLOCK "IO_Valve_Blend20_DB"   // DB28
VERSION : 0.1
// stored: AutoNumber true, DBAccessibleFromOPCUA true, DBAccessibleFromWebserver true, InstanceOfName IO_Valve_Blend20, InstanceOfType FB
"IO_Valve_Blend20"
BEGIN
END_DATA_BLOCK

DATA_BLOCK "IO_Valve_Blend21_DB"   // DB39
VERSION : 0.1
// stored: AutoNumber true, DBAccessibleFromOPCUA true, DBAccessibleFromWebserver true, InstanceOfName IO_Valve_Blend21, InstanceOfType FB
"IO_Valve_Blend21"
BEGIN
END_DATA_BLOCK

DATA_BLOCK "IO_Valve_Blend30_DB"   // DB60
VERSION : 0.1
// stored: AutoNumber true, DBAccessibleFromOPCUA true, DBAccessibleFromWebserver true, InstanceOfName IO_Valve_Blend30, InstanceOfType FB
"IO_Valve_Blend30"
BEGIN
END_DATA_BLOCK

DATA_BLOCK "IO_Valve_Blend31_DB"   // DB61
VERSION : 0.1
// stored: AutoNumber true, DBAccessibleFromOPCUA true, DBAccessibleFromWebserver true, InstanceOfName IO_Valve_Blend31, InstanceOfType FB
"IO_Valve_Blend31"
BEGIN
END_DATA_BLOCK

DATA_BLOCK "IO_Valve_Blend40_DB"   // DB26
VERSION : 0.1
// stored: AutoNumber true, DBAccessibleFromOPCUA true, DBAccessibleFromWebserver true, InstanceOfName IO_Valve_Blend40, InstanceOfType FB
"IO_Valve_Blend40"
BEGIN
END_DATA_BLOCK

DATA_BLOCK "IO_Valve_Blend41_DB"   // DB62
VERSION : 0.1
// stored: AutoNumber true, DBAccessibleFromOPCUA true, DBAccessibleFromWebserver true, InstanceOfName IO_Valve_Blend41, InstanceOfType FB
"IO_Valve_Blend41"
BEGIN
END_DATA_BLOCK

DATA_BLOCK "IO_Valve_Blending_DB"   // DB8
VERSION : 0.1
// stored: AutoNumber true, DBAccessibleFromOPCUA true, DBAccessibleFromWebserver true, InstanceOfName IO_Valve_Blending, InstanceOfType FB
"IO_Valve_Blending"
BEGIN
   "AV-20.02".OPdwCmd := 16#0008_0000;
   "AV-20.03".OPdwCmd := 16#0008_0000;
   "AV-20.04".OPdwCmd := 16#0008_0000;
   "AV-20.05".OPdwCmd := 16#0008_0000;
   "AV-20.06".OPdwCmd := 16#0008_0000;
   "AV-20.07".OPdwCmd := 16#0008_0000;
   "AV-20.08".OPdwCmd := 16#0008_0000;
   "AV-20.09".OPdwCmd := 16#0008_0000;
   "AV-20.10".OPdwCmd := 16#0008_0000;
   "AV-20.11".OPdwCmd := 16#0008_0000;
   "AV-20.12".OPdwCmd := 16#0008_0000;
   "AV-20.13".OPdwCmd := 16#0008_0000;
   "AV-20.14".OPdwCmd := 16#0008_0000;
   "AV-20.15".OPdwCmd := 16#0008_0000;
   "AV-20.16".OPdwCmd := 16#0008_0000;
   "AV-20.17".OPdwCmd := 16#0008_0000;
   "AV-20.31".OPdwCmd := 16#0008_0000;
   "AV-20.32".OPdwCmd := 16#0008_0000;
   "AV-20.33".OPdwCmd := 16#0008_0000;
   "AV-20.34".OPdwCmd := 16#0008_0000;
   "AV-20.35".OPdwCmd := 16#0008_0000;
   "AV-20.36".OPdwCmd := 16#0008_0000;
   "AV-20.37".OPdwCmd := 16#0008_0000;
   "AV-20.38".OPdwCmd := 16#0008_0000;
   "AV-20.39".OPdwCmd := 16#0008_0000;
   "AV-20.40".OPdwCmd := 16#0008_0000;
   "AV-20.41".OPdwCmd := 16#0008_0000;
   "AV-21.01".OPdwCmd := 16#0008_0000;
   "AV-21.02".OPdwCmd := 16#0008_0000;
   "AV-21.03".OPdwCmd := 16#0008_0000;
   "AV-21.04".OPdwCmd := 16#0008_0000;
   "AV-21.05".OPdwCmd := 16#0008_0000;
   "AV-21.06".OPdwCmd := 16#0008_0000;
   "AV-21.07".OPdwCmd := 16#0008_0000;
   "AV-21.08".OPdwCmd := 16#0008_0000;
   "AV-21.09".OPdwCmd := 16#0008_0000;
   "AV-21.10".OPdwCmd := 16#0008_0000;
   "AV-21.11".OPdwCmd := 16#0008_0000;
   "AV-21.12".OPdwCmd := 16#0008_0000;
   "AV-21.13".OPdwCmd := 16#0008_0000;
   "AV-21.14".OPdwCmd := 16#0008_0000;
   "AV-21.15".OPdwCmd := 16#0008_0000;
   "AV-21.16".OPdwCmd := 16#0008_0000;
   "AV-21.17".OPdwCmd := 16#0008_0000;
   "AV-21.18".OPdwCmd := 16#0008_0000;
   "AV-21.31".OPdwCmd := 16#0008_0000;
   "AV-21.32".OPdwCmd := 16#0008_0000;
   "AV-21.33".OPdwCmd := 16#0008_0000;
   "AV-21.34".OPdwCmd := 16#0008_0000;
   "AV-21.35".OPdwCmd := 16#0008_0000;
   "AV-21.36".OPdwCmd := 16#0008_0000;
   "AV-21.37".OPdwCmd := 16#0008_0000;
   "AV-21.38".OPdwCmd := 16#0008_0000;
   "AV-21.39".OPdwCmd := 16#0008_0000;
   "AV-21.40".OPdwCmd := 16#0008_0000;
   "AV-21.41".OPdwCmd := 16#0008_0000;
   "AV-22.01".OPdwCmd := 16#0008_0000;
   "AV-22.02".OPdwCmd := 16#0008_0000;
   "AV-22.03".OPdwCmd := 16#0008_0000;
   "AV-22.06".OPdwCmd := 16#0008_0000;
   "AV-22.11".OPdwCmd := 16#0008_0000;
   "AV-22.21".OPdwCmd := 16#0008_0000;
   "AV-22.22".OPdwCmd := 16#0008_0000;
   "AV-30.01".OPdwCmd := 16#0008_0000;
   "AV-30.02".OPdwCmd := 16#0008_0000;
   "AV-30.03".OPdwCmd := 16#0008_0000;
   "AV-30.04".OPdwCmd := 16#0008_0000;
   "AV-30.05".OPdwCmd := 16#0008_0000;
   "AV-30.06".OPdwCmd := 16#0008_0000;
   "AV-30.07".OPdwCmd := 16#0008_0000;
   "AV-30.08".OPdwCmd := 16#0008_0000;
   "AV-30.09".OPdwCmd := 16#0008_0000;
   "AV-30.10".OPdwCmd := 16#0008_0000;
   "AV-30.11".OPdwCmd := 16#0008_0000;
   "AV-30.12".OPdwCmd := 16#0008_0000;
   "AV-30.13".OPdwCmd := 16#0008_0000;
   "AV-30.14".OPdwCmd := 16#0008_0000;
   "AV-30.15".OPdwCmd := 16#0008_0000;
   "AV-30.16".OPdwCmd := 16#0008_0000;
   "AV-30.17".OPdwCmd := 16#0008_0000;
   "AV-30.31".OPdwCmd := 16#0008_0000;
   "AV-30.32".OPdwCmd := 16#0008_0000;
   "AV-30.33".OPdwCmd := 16#0008_0000;
   "AV-30.34".OPdwCmd := 16#0008_0000;
   "AV-30.35".OPdwCmd := 16#0008_0000;
   "AV-30.36".OPdwCmd := 16#0008_0000;
   "AV-30.37".OPdwCmd := 16#0008_0000;
   "AV-30.38".OPdwCmd := 16#0008_0000;
   "AV-30.39".OPdwCmd := 16#0008_0000;
   "AV-30.40".OPdwCmd := 16#0008_0000;
   "AV-30.41".OPdwCmd := 16#0008_0000;
   "AV-31.01".OPdwCmd := 16#0008_0000;
   "AV-31.02".OPdwCmd := 16#0008_0000;
   "AV-31.03".OPdwCmd := 16#0008_0000;
   "AV-31.04".OPdwCmd := 16#0008_0000;
   "AV-31.05".OPdwCmd := 16#0008_0000;
   "AV-31.06".OPdwCmd := 16#0008_0000;
   "AV-31.07".OPdwCmd := 16#0008_0000;
   "AV-31.08".OPdwCmd := 16#0008_0000;
   "AV-31.09".OPdwCmd := 16#0008_0000;
   "AV-31.10".OPdwCmd := 16#0008_0000;
   "AV-31.11".OPdwCmd := 16#0008_0000;
   "AV-31.12".OPdwCmd := 16#0008_0000;
   "AV-31.13".OPdwCmd := 16#0008_0000;
   "AV-31.14".OPdwCmd := 16#0008_0000;
   "AV-31.15".OPdwCmd := 16#0008_0000;
   "AV-31.16".OPdwCmd := 16#0008_0000;
   "AV-31.17".OPdwCmd := 16#0008_0000;
   "AV-31.18".OPdwCmd := 16#0008_0000;
   "AV-31.31".OPdwCmd := 16#0008_0000;
   "AV-31.32".OPdwCmd := 16#0008_0000;
   "AV-31.33".OPdwCmd := 16#0008_0000;
   "AV-31.34".OPdwCmd := 16#0008_0000;
   "AV-31.35".OPdwCmd := 16#0008_0000;
   "AV-31.36".OPdwCmd := 16#0008_0000;
   "AV-31.37".OPdwCmd := 16#0008_0000;
   "AV-31.38".OPdwCmd := 16#0008_0000;
   "AV-31.39".OPdwCmd := 16#0008_0000;
   "AV-31.40".OPdwCmd := 16#0008_0000;
   "AV-31.41".OPdwCmd := 16#0008_0000;
   "AV-31.51".OPdwCmd := 16#0008_0000;
   "AV-31.52".OPdwCmd := 16#0008_0000;
   "AV-31.53".OPdwCmd := 16#0008_0000;
   "AV-31.54".OPdwCmd := 16#0008_0000;
   "AV-31.55".OPdwCmd := 16#0008_0000;
   "AV-31.56".OPdwCmd := 16#0008_0000;
   "AV-31.57".OPdwCmd := 16#0008_0000;
   "AV-31.58".OPdwCmd := 16#0008_0000;
   "AV-31.59".OPdwCmd := 16#0008_0000;
   "AV-31.60".OPdwCmd := 16#0008_0000;
   "AV-31.61".OPdwCmd := 16#0008_0000;
   "AV-31.62".OPdwCmd := 16#0008_0000;
   "AV-32.01".OPdwCmd := 16#0008_0000;
   "AV-32.02".OPdwCmd := 16#0008_0000;
   "AV-32.03".OPdwCmd := 16#0008_0000;
   "AV-32.06".OPdwCmd := 16#0008_0000;
   "AV-32.11".OPdwCmd := 16#0008_0000;
   "AV-32.21".OPdwCmd := 16#0008_0000;
   "AV-32.22".OPdwCmd := 16#0008_0000;
   "AV-20.42".OPdwCmd := 16#0008_0000;
   "AV-21.42".OPdwCmd := 16#0008_0000;
   "AV-22.04".OPdwCmd := 16#0008_0000;
   "AV-22.05".OPdwCmd := 16#0008_0000;
   "AV-30.42".OPdwCmd := 16#0008_0000;
   "AV-31.42".OPdwCmd := 16#0008_0000;
   "AV-32.04".OPdwCmd := 16#0008_0000;
   "AV-32.05".OPdwCmd := 16#0008_0000;
END_DATA_BLOCK

DATA_BLOCK "IO Analog Storage_DB"   // DB9
VERSION : 0.1
// stored: AutoNumber true, DBAccessibleFromOPCUA true, DBAccessibleFromWebserver true, InstanceOfName IO Analog Storage, InstanceOfType FB
"IO Analog Storage"
BEGIN
END_DATA_BLOCK

DATA_BLOCK "IO_Digital_Storage_DB"   // DB44
VERSION : 0.1
// stored: AutoNumber true, DBAccessibleFromOPCUA true, DBAccessibleFromWebserver true, InstanceOfName IO_Digital_Storage, InstanceOfType FB
"IO_Digital_Storage"
BEGIN
END_DATA_BLOCK

DATA_BLOCK "IO_Valve_Storage_DB"   // DB11
VERSION : 0.1
// stored: AutoNumber true, DBAccessibleFromOPCUA true, DBAccessibleFromWebserver true, InstanceOfName IO_Valve_Storage, InstanceOfType FB
"IO_Valve_Storage"
BEGIN
END_DATA_BLOCK

DATA_BLOCK "IO Motor MCC Preparation_DB"   // DB12
VERSION : 0.1
// stored: AutoNumber true, DBAccessibleFromOPCUA true, DBAccessibleFromWebserver true, InstanceOfName IO Motor MCC Preparation, InstanceOfType FB
"IO Motor MCC Preparation"
BEGIN
END_DATA_BLOCK

DATA_BLOCK "IO Analog Preparation_DB"   // DB13
VERSION : 0.1
// stored: AutoNumber true, DBAccessibleFromOPCUA true, DBAccessibleFromWebserver true, InstanceOfName IO Analog Preparation, InstanceOfType FB
"IO Analog Preparation"
BEGIN
END_DATA_BLOCK

DATA_BLOCK "IO Digital Preparation_DB"   // DB14
VERSION : 0.1
// stored: AutoNumber true, DBAccessibleFromOPCUA true, DBAccessibleFromWebserver true, InstanceOfName IO Digital Preparation, InstanceOfType FB
"IO Digital Preparation"
BEGIN
END_DATA_BLOCK

DATA_BLOCK "IO_Valve_T01_HWT"   // DB301
VERSION : 0.1
// stored: AutoNumber false, DBAccessibleFromOPCUA true, DBAccessibleFromWebserver true, InstanceOfName IO Valve T01 HWT, InstanceOfType FB
"IO Valve T01 HWT"
BEGIN
END_DATA_BLOCK

DATA_BLOCK "IO_Valve_T02_Chili"   // DB302
VERSION : 0.1
// stored: AutoNumber false, DBAccessibleFromOPCUA true, DBAccessibleFromWebserver true, InstanceOfName IO Valve T02 Chili, InstanceOfType FB
"IO Valve T02 Chili"
BEGIN
END_DATA_BLOCK

DATA_BLOCK "IO_Valve_T03_Chili"   // DB303
VERSION : 0.1
// stored: AutoNumber false, DBAccessibleFromOPCUA true, DBAccessibleFromWebserver true, InstanceOfName IO Valve T03 Chili, InstanceOfType FB
"IO Valve T03 Chili"
BEGIN
END_DATA_BLOCK

DATA_BLOCK "IO_Valve_T04_Chili"   // DB304
VERSION : 0.1
// stored: AutoNumber false, DBAccessibleFromOPCUA true, DBAccessibleFromWebserver true, InstanceOfName IO Valve T04 Chili, InstanceOfType FB
"IO Valve T04 Chili"
BEGIN
END_DATA_BLOCK

DATA_BLOCK "IO_Valve_T05_Tomato"   // DB305
VERSION : 0.1
// stored: AutoNumber false, DBAccessibleFromOPCUA true, DBAccessibleFromWebserver true, InstanceOfName IO Valve T05 Tomato, InstanceOfType FB
"IO Valve T05 Tomato"
BEGIN
END_DATA_BLOCK

DATA_BLOCK "IO_Valve_T06_FreshChili"   // DB306
VERSION : 0.1
// stored: AutoNumber false, DBAccessibleFromOPCUA true, DBAccessibleFromWebserver true, InstanceOfName IO Valve T06 FreshChili, InstanceOfType FB
"IO Valve T06 FreshChili"
BEGIN
END_DATA_BLOCK

DATA_BLOCK "IO_Valve_T07_FreshChili"   // DB307
VERSION : 0.1
// stored: AutoNumber false, DBAccessibleFromOPCUA true, DBAccessibleFromWebserver true, InstanceOfName IO Valve T07 FreshChili, InstanceOfType FB
"IO Valve T07 FreshChili"
BEGIN
END_DATA_BLOCK

DATA_BLOCK "IO_Valve_T08_FreshChili"   // DB308
VERSION : 0.1
// stored: AutoNumber false, DBAccessibleFromOPCUA true, DBAccessibleFromWebserver true, InstanceOfName IO Valve T08 FreshChili, InstanceOfType FB
"IO Valve T08 FreshChili"
BEGIN
END_DATA_BLOCK

DATA_BLOCK "IO_Valve_T09_Garlic"   // DB309
VERSION : 0.1
// stored: AutoNumber false, DBAccessibleFromOPCUA true, DBAccessibleFromWebserver true, InstanceOfName IO Valve T09 Garlic, InstanceOfType FB
"IO Valve T09 Garlic"
BEGIN
END_DATA_BLOCK

DATA_BLOCK "IO_Valve_T10_Vinegar"   // DB310
VERSION : 0.1
// stored: AutoNumber false, DBAccessibleFromOPCUA true, DBAccessibleFromWebserver true, InstanceOfName IO Valve T10 Vinegar, InstanceOfType FB
"IO Valve T10 Vinegar"
BEGIN
END_DATA_BLOCK

DATA_BLOCK "IO_Valve_T51_HW"   // DB311
VERSION : 0.1
// stored: AutoNumber false, DBAccessibleFromOPCUA true, DBAccessibleFromWebserver true, InstanceOfName IO Valve T51 HotWaterLine, InstanceOfType FB
"IO Valve T51 HotWaterLine"
BEGIN
END_DATA_BLOCK

DATA_BLOCK "IO_Valve_Buffer_DB"   // DB64
VERSION : 0.1
// stored: AutoNumber true, DBAccessibleFromOPCUA true, DBAccessibleFromWebserver true, InstanceOfName IO_Valve_Buffer, InstanceOfType FB
"IO_Valve_Buffer"
BEGIN
END_DATA_BLOCK

DATA_BLOCK "Totalizer_FT-00.01"   // DB381
VERSION : 0.1
// stored: AutoNumber false, DBAccessibleFromOPCUA true, DBAccessibleFromWebserver true, InstanceOfName Totalizer, InstanceOfType FB
"Totalizer"
   // VAR_INPUT
   //    value : Real;
   //    intervall : Time;
   //    cycle : Time;
   //    reset : Bool;
   // END_VAR
   // VAR_OUTPUT
   //    total : Real;
   // END_VAR
   // VAR
   //    statAccum : Real;
   // END_VAR
BEGIN
END_DATA_BLOCK

DATA_BLOCK "Totalizer_FT-02.01"   // DB382
VERSION : 0.1
// stored: AutoNumber false, DBAccessibleFromOPCUA true, DBAccessibleFromWebserver true, InstanceOfName Totalizer, InstanceOfType FB
"Totalizer"
   // VAR_INPUT
   //    value : Real;
   //    intervall : Time;
   //    cycle : Time;
   //    reset : Bool;
   // END_VAR
   // VAR_OUTPUT
   //    total : Real;
   // END_VAR
   // VAR
   //    statAccum : Real;
   // END_VAR
BEGIN
END_DATA_BLOCK

DATA_BLOCK "Totalizer_FT-03.01"   // DB383
VERSION : 0.1
// stored: AutoNumber false, DBAccessibleFromOPCUA true, DBAccessibleFromWebserver true, InstanceOfName Totalizer, InstanceOfType FB
"Totalizer"
   // VAR_INPUT
   //    value : Real;
   //    intervall : Time;
   //    cycle : Time;
   //    reset : Bool;
   // END_VAR
   // VAR_OUTPUT
   //    total : Real;
   // END_VAR
   // VAR
   //    statAccum : Real;
   // END_VAR
BEGIN
END_DATA_BLOCK

DATA_BLOCK "Totalizer_FT-04.01"   // DB384
VERSION : 0.1
// stored: AutoNumber false, DBAccessibleFromOPCUA true, DBAccessibleFromWebserver true, InstanceOfName Totalizer, InstanceOfType FB
"Totalizer"
   // VAR_INPUT
   //    value : Real;
   //    intervall : Time;
   //    cycle : Time;
   //    reset : Bool;
   // END_VAR
   // VAR_OUTPUT
   //    total : Real;
   // END_VAR
   // VAR
   //    statAccum : Real;
   // END_VAR
BEGIN
END_DATA_BLOCK

DATA_BLOCK "Totalizer_FT-05.01"   // DB385
VERSION : 0.1
// stored: AutoNumber false, DBAccessibleFromOPCUA true, DBAccessibleFromWebserver true, InstanceOfName Totalizer, InstanceOfType FB
"Totalizer"
   // VAR_INPUT
   //    value : Real;
   //    intervall : Time;
   //    cycle : Time;
   //    reset : Bool;
   // END_VAR
   // VAR_OUTPUT
   //    total : Real;
   // END_VAR
   // VAR
   //    statAccum : Real;
   // END_VAR
BEGIN
END_DATA_BLOCK

DATA_BLOCK "Totalizer_FT-06.01"   // DB386
VERSION : 0.1
// stored: AutoNumber false, DBAccessibleFromOPCUA true, DBAccessibleFromWebserver true, InstanceOfName Totalizer, InstanceOfType FB
"Totalizer"
   // VAR_INPUT
   //    value : Real;
   //    intervall : Time;
   //    cycle : Time;
   //    reset : Bool;
   // END_VAR
   // VAR_OUTPUT
   //    total : Real;
   // END_VAR
   // VAR
   //    statAccum : Real;
   // END_VAR
BEGIN
END_DATA_BLOCK

DATA_BLOCK "Totalizer_FT-07.01"   // DB387
VERSION : 0.1
// stored: AutoNumber false, DBAccessibleFromOPCUA true, DBAccessibleFromWebserver true, InstanceOfName Totalizer, InstanceOfType FB
"Totalizer"
   // VAR_INPUT
   //    value : Real;
   //    intervall : Time;
   //    cycle : Time;
   //    reset : Bool;
   // END_VAR
   // VAR_OUTPUT
   //    total : Real;
   // END_VAR
   // VAR
   //    statAccum : Real;
   // END_VAR
BEGIN
END_DATA_BLOCK

DATA_BLOCK "Totalizer_FT-08.01"   // DB388
VERSION : 0.1
// stored: AutoNumber false, DBAccessibleFromOPCUA true, DBAccessibleFromWebserver true, InstanceOfName Totalizer, InstanceOfType FB
"Totalizer"
   // VAR_INPUT
   //    value : Real;
   //    intervall : Time;
   //    cycle : Time;
   //    reset : Bool;
   // END_VAR
   // VAR_OUTPUT
   //    total : Real;
   // END_VAR
   // VAR
   //    statAccum : Real;
   // END_VAR
BEGIN
END_DATA_BLOCK

DATA_BLOCK "Totalizer_FT-09.01"   // DB389
VERSION : 0.1
// stored: AutoNumber false, DBAccessibleFromOPCUA true, DBAccessibleFromWebserver true, InstanceOfName Totalizer, InstanceOfType FB
"Totalizer"
   // VAR_INPUT
   //    value : Real;
   //    intervall : Time;
   //    cycle : Time;
   //    reset : Bool;
   // END_VAR
   // VAR_OUTPUT
   //    total : Real;
   // END_VAR
   // VAR
   //    statAccum : Real;
   // END_VAR
BEGIN
END_DATA_BLOCK

DATA_BLOCK "Totalizer_FT-10.01"   // DB390
VERSION : 0.1
// stored: AutoNumber false, DBAccessibleFromOPCUA true, DBAccessibleFromWebserver true, InstanceOfName Totalizer, InstanceOfType FB
"Totalizer"
   // VAR_INPUT
   //    value : Real;
   //    intervall : Time;
   //    cycle : Time;
   //    reset : Bool;
   // END_VAR
   // VAR_OUTPUT
   //    total : Real;
   // END_VAR
   // VAR
   //    statAccum : Real;
   // END_VAR
BEGIN
END_DATA_BLOCK

DATA_BLOCK "Totalizer_FT-12.01"   // DB393
VERSION : 0.1
// stored: AutoNumber false, DBAccessibleFromOPCUA true, DBAccessibleFromWebserver true, InstanceOfName Totalizer, InstanceOfType FB
"Totalizer"
   // VAR_INPUT
   //    value : Real;
   //    intervall : Time;
   //    cycle : Time;
   //    reset : Bool;
   // END_VAR
   // VAR_OUTPUT
   //    total : Real;
   // END_VAR
   // VAR
   //    statAccum : Real;
   // END_VAR
BEGIN
END_DATA_BLOCK

DATA_BLOCK "Totalizer_FT-12.02"   // DB394
VERSION : 0.1
// stored: AutoNumber false, DBAccessibleFromOPCUA true, DBAccessibleFromWebserver true, InstanceOfName Totalizer, InstanceOfType FB
"Totalizer"
   // VAR_INPUT
   //    value : Real;
   //    intervall : Time;
   //    cycle : Time;
   //    reset : Bool;
   // END_VAR
   // VAR_OUTPUT
   //    total : Real;
   // END_VAR
   // VAR
   //    statAccum : Real;
   // END_VAR
BEGIN
END_DATA_BLOCK

DATA_BLOCK "Totalizer_FT-51.01"   // DB391
VERSION : 0.1
// stored: AutoNumber false, DBAccessibleFromOPCUA true, DBAccessibleFromWebserver true, InstanceOfName Totalizer, InstanceOfType FB
"Totalizer"
   // VAR_INPUT
   //    value : Real;
   //    intervall : Time;
   //    cycle : Time;
   //    reset : Bool;
   // END_VAR
   // VAR_OUTPUT
   //    total : Real;
   // END_VAR
   // VAR
   //    statAccum : Real;
   // END_VAR
BEGIN
END_DATA_BLOCK

DATA_BLOCK "GET_DB_1"   // DB27
// stored: AutoNumber true, DBAccessibleFromOPCUA true, DBAccessibleFromWebserver true, InstanceOfName GET_SFB, OfSystemLibElement GET, OfSystemLibVersion 1.2
"GET_SFB"
   // VAR_INPUT
   //    REQ : Bool;
   //    ID : Word;
   // END_VAR
   // VAR_OUTPUT
   //    NDR : Bool;
   //    ERROR : Bool;
   //    STATUS : Word;
   // END_VAR
   // VAR_IN_OUT
   //    ADDR_1 : Remote;
   //    ADDR_2 : Remote;
   //    ADDR_3 : Remote;
   //    ADDR_4 : Remote;
   //    RD_1 : Variant;
   //    RD_2 : Variant;
   //    RD_3 : Variant;
   //    RD_4 : Variant;
   // END_VAR
BEGIN
END_DATA_BLOCK

DATA_BLOCK "GET_OSA_CIP"   // DB50
// stored: AutoNumber false, DBAccessibleFromOPCUA true, DBAccessibleFromWebserver true, InstanceOfName GET_SFB, OfSystemLibElement GET, OfSystemLibVersion 1.2
"GET_SFB"
   // VAR_INPUT
   //    REQ : Bool;
   //    ID : Word;
   // END_VAR
   // VAR_OUTPUT
   //    NDR : Bool;
   //    ERROR : Bool;
   //    STATUS : Word;
   // END_VAR
   // VAR_IN_OUT
   //    ADDR_1 : Remote;
   //    ADDR_2 : Remote;
   //    ADDR_3 : Remote;
   //    ADDR_4 : Remote;
   //    RD_1 : Variant;
   //    RD_2 : Variant;
   //    RD_3 : Variant;
   //    RD_4 : Variant;
   // END_VAR
BEGIN
END_DATA_BLOCK

DATA_BLOCK "GET_OSA_Chili"   // DB57
// stored: AutoNumber false, DBAccessibleFromOPCUA true, DBAccessibleFromWebserver true, InstanceOfName GET_SFB, OfSystemLibElement GET, OfSystemLibVersion 1.2
"GET_SFB"
   // VAR_INPUT
   //    REQ : Bool;
   //    ID : Word;
   // END_VAR
   // VAR_OUTPUT
   //    NDR : Bool;
   //    ERROR : Bool;
   //    STATUS : Word;
   // END_VAR
   // VAR_IN_OUT
   //    ADDR_1 : Remote;
   //    ADDR_2 : Remote;
   //    ADDR_3 : Remote;
   //    ADDR_4 : Remote;
   //    RD_1 : Variant;
   //    RD_2 : Variant;
   //    RD_3 : Variant;
   //    RD_4 : Variant;
   // END_VAR
BEGIN
END_DATA_BLOCK

DATA_BLOCK "Get_Tipper1"   // DB242
// stored: AutoNumber false, DBAccessibleFromOPCUA true, DBAccessibleFromWebserver true, InstanceOfName GET_SFB, OfSystemLibElement GET, OfSystemLibVersion 1.2
"GET_SFB"
   // VAR_INPUT
   //    REQ : Bool;
   //    ID : Word;
   // END_VAR
   // VAR_OUTPUT
   //    NDR : Bool;
   //    ERROR : Bool;
   //    STATUS : Word;
   // END_VAR
   // VAR_IN_OUT
   //    ADDR_1 : Remote;
   //    ADDR_2 : Remote;
   //    ADDR_3 : Remote;
   //    ADDR_4 : Remote;
   //    RD_1 : Variant;
   //    RD_2 : Variant;
   //    RD_3 : Variant;
   //    RD_4 : Variant;
   // END_VAR
BEGIN
END_DATA_BLOCK

DATA_BLOCK "Get_Tipper2"   // DB246
// stored: AutoNumber false, DBAccessibleFromOPCUA true, DBAccessibleFromWebserver true, InstanceOfName GET_SFB, OfSystemLibElement GET, OfSystemLibVersion 1.2
"GET_SFB"
   // VAR_INPUT
   //    REQ : Bool;
   //    ID : Word;
   // END_VAR
   // VAR_OUTPUT
   //    NDR : Bool;
   //    ERROR : Bool;
   //    STATUS : Word;
   // END_VAR
   // VAR_IN_OUT
   //    ADDR_1 : Remote;
   //    ADDR_2 : Remote;
   //    ADDR_3 : Remote;
   //    ADDR_4 : Remote;
   //    RD_1 : Variant;
   //    RD_2 : Variant;
   //    RD_3 : Variant;
   //    RD_4 : Variant;
   // END_VAR
BEGIN
END_DATA_BLOCK

DATA_BLOCK "PUT_OSA_CIP"   // DB56
// stored: AutoNumber false, DBAccessibleFromOPCUA true, DBAccessibleFromWebserver true, InstanceOfName PUT_SFB, OfSystemLibElement PUT, OfSystemLibVersion 1.3
"PUT_SFB"
   // VAR_INPUT
   //    REQ : Bool;
   //    ID : Word;
   // END_VAR
   // VAR_OUTPUT
   //    DONE : Bool;
   //    ERROR : Bool;
   //    STATUS : Word;
   // END_VAR
   // VAR_IN_OUT
   //    ADDR_1 : Remote;
   //    ADDR_2 : Remote;
   //    ADDR_3 : Remote;
   //    ADDR_4 : Remote;
   //    SD_1 : Variant;
   //    SD_2 : Variant;
   //    SD_3 : Variant;
   //    SD_4 : Variant;
   // END_VAR
BEGIN
END_DATA_BLOCK

DATA_BLOCK "PUT_OSA_Chili"   // DB58
// stored: AutoNumber true, DBAccessibleFromOPCUA true, DBAccessibleFromWebserver true, InstanceOfName PUT_SFB, OfSystemLibElement PUT, OfSystemLibVersion 1.3
"PUT_SFB"
   // VAR_INPUT
   //    REQ : Bool;
   //    ID : Word;
   // END_VAR
   // VAR_OUTPUT
   //    DONE : Bool;
   //    ERROR : Bool;
   //    STATUS : Word;
   // END_VAR
   // VAR_IN_OUT
   //    ADDR_1 : Remote;
   //    ADDR_2 : Remote;
   //    ADDR_3 : Remote;
   //    ADDR_4 : Remote;
   //    SD_1 : Variant;
   //    SD_2 : Variant;
   //    SD_3 : Variant;
   //    SD_4 : Variant;
   // END_VAR
BEGIN
END_DATA_BLOCK

DATA_BLOCK "Put_Tipper1"   // DB243
// stored: AutoNumber false, DBAccessibleFromOPCUA true, DBAccessibleFromWebserver true, InstanceOfName PUT_SFB, OfSystemLibElement PUT, OfSystemLibVersion 1.3
"PUT_SFB"
   // VAR_INPUT
   //    REQ : Bool;
   //    ID : Word;
   // END_VAR
   // VAR_OUTPUT
   //    DONE : Bool;
   //    ERROR : Bool;
   //    STATUS : Word;
   // END_VAR
   // VAR_IN_OUT
   //    ADDR_1 : Remote;
   //    ADDR_2 : Remote;
   //    ADDR_3 : Remote;
   //    ADDR_4 : Remote;
   //    SD_1 : Variant;
   //    SD_2 : Variant;
   //    SD_3 : Variant;
   //    SD_4 : Variant;
   // END_VAR
BEGIN
END_DATA_BLOCK

DATA_BLOCK "Put_Tipper2"   // DB247
// stored: AutoNumber false, DBAccessibleFromOPCUA true, DBAccessibleFromWebserver true, InstanceOfName PUT_SFB, OfSystemLibElement PUT, OfSystemLibVersion 1.3
"PUT_SFB"
   // VAR_INPUT
   //    REQ : Bool;
   //    ID : Word;
   // END_VAR
   // VAR_OUTPUT
   //    DONE : Bool;
   //    ERROR : Bool;
   //    STATUS : Word;
   // END_VAR
   // VAR_IN_OUT
   //    ADDR_1 : Remote;
   //    ADDR_2 : Remote;
   //    ADDR_3 : Remote;
   //    ADDR_4 : Remote;
   //    SD_1 : Variant;
   //    SD_2 : Variant;
   //    SD_3 : Variant;
   //    SD_4 : Variant;
   // END_VAR
BEGIN
END_DATA_BLOCK

DATA_BLOCK "Timer_Pulse_Drain_Water_THE1"   // DB30
{ S7_Optimized_Access := 'TRUE' }
// stored: AutoNumber true, DBAccessibleFromOPCUA true, DBAccessibleFromWebserver true, InstanceOfName IEC_TIMER, OfSystemLibElement IEC_TIMER, OfSystemLibVersion 1.0
"IEC_TIMER"
   // VAR
   //    PT : Time := T#15s;
   //    ET { ExternalWritable := 'False'} : Time;
   //    IN : Bool;
   //    Q { ExternalWritable := 'False'} : Bool;
   // END_VAR
BEGIN
END_DATA_BLOCK

DATA_BLOCK "Timer_Pulse_Drain_Water_THE2"   // DB29
{ S7_Optimized_Access := 'TRUE' }
// stored: AutoNumber true, DBAccessibleFromOPCUA true, DBAccessibleFromWebserver true, InstanceOfName IEC_TIMER, OfSystemLibElement IEC_TIMER, OfSystemLibVersion 1.0
"IEC_TIMER"
   // VAR
   //    PT : Time := T#15s;
   //    ET { ExternalWritable := 'False'} : Time;
   //    IN : Bool;
   //    Q { ExternalWritable := 'False'} : Bool;
   // END_VAR
BEGIN
END_DATA_BLOCK

DATA_BLOCK "Rework_T-22_DB"   // DB48
VERSION : 0.1
// stored: AutoNumber false, DBAccessibleFromOPCUA true, DBAccessibleFromWebserver true, InstanceOfName Rework, InstanceOfType FB
"Rework"
BEGIN
END_DATA_BLOCK

DATA_BLOCK "Rework_T-32_DB"   // DB49
VERSION : 0.1
// stored: AutoNumber false, DBAccessibleFromOPCUA true, DBAccessibleFromWebserver true, InstanceOfName Rework, InstanceOfType FB
"Rework"
BEGIN
END_DATA_BLOCK

DATA_BLOCK "T-20.00_DB"   // DB18
VERSION : 0.1
// stored: AutoNumber true, DBAccessibleFromOPCUA true, DBAccessibleFromWebserver true, InstanceOfName BLEND, InstanceOfType FB
"BLEND"
BEGIN
END_DATA_BLOCK

DATA_BLOCK "T-21.00_DB"   // DB19
VERSION : 0.1
// stored: AutoNumber true, DBAccessibleFromOPCUA true, DBAccessibleFromWebserver true, InstanceOfName BLEND, InstanceOfType FB
"BLEND"
BEGIN
END_DATA_BLOCK

DATA_BLOCK "T-30.00_DB"   // DB24
VERSION : 0.1
// stored: AutoNumber true, DBAccessibleFromOPCUA true, DBAccessibleFromWebserver true, InstanceOfName BLEND, InstanceOfType FB
"BLEND"
BEGIN
END_DATA_BLOCK

DATA_BLOCK "T-31.00_DB"   // DB25
VERSION : 0.1
// stored: AutoNumber true, DBAccessibleFromOPCUA true, DBAccessibleFromWebserver true, InstanceOfName BLEND, InstanceOfType FB
"BLEND"
BEGIN
END_DATA_BLOCK

DATA_BLOCK "T-01.01_DB"   // DB351
VERSION : 0.1
// stored: AutoNumber false, DBAccessibleFromOPCUA true, DBAccessibleFromWebserver true, InstanceOfName HWT, InstanceOfType FB
"HWT"
   // VAR_INPUT
   //    "IN_FBAV.01" : Bool;
   //    "IN_FBAV.02" : Bool;
   //    "IN_FBAV.03" : Bool;
   //    "IN_FBAV.04" : Bool;
   //    "IN_FBAV.10" : Bool;
   //    "IN_FBCV.10" : Bool;
   //    "IN_FS.01" : Bool;
   //    IN_LT01 : Real;
   //    IN_TT01 : Real;
   //    IN_TT02 : Real;
   //    "IN_FBP.01" : Bool;
   //    "IN_P.01-Speed" : Real;
   //    DosePumpSpeed : Real;
   //    "DoseON-OFF" : Bool;
   //    "DosePumpON-OFF" : Bool;
   //    CIPPulse : Bool;
   //    Line_OK : Bool;
   // END_VAR
   // VAR_OUTPUT
   //    "OUT_AV.01" : Bool;
   //    "OUT_AV.02" : Bool;
   //    "OUT_AV.03" : Bool;
   //    "OUT_AV.04" : Bool;
   //    "OUT_AV.10" : Bool;
   //    "OUT_CV.10" : Bool;
   //    Q_PID_Setpoint : Real;
   //    Q_PID_PV_IN : Real;
   //    "OUT_FS.01" : Bool;
   //    "OUT_LT.01" : Real;
   //    "OUT_TT.01" : Real;
   //    "OUT_TT.02" : Real;
   //    "OUT_P.01" : Bool;
   //    "OUT_P.01-Speed" : Real;
   //    OUT_CIP_Request : Bool;
   //    Q_WH_Tank_Ready : Bool;
   // END_VAR
   // VAR
   //    Cmd : Struct
   //       Start_Prosses : Bool;
   //       Start_Preheat : Bool;
   //       HWT_Mode : Bool;
   //       Ready_for_Mix : Bool;
   //       "CIP Request" : Bool;
   //       Pump_Mode : Bool;
   //       Pump_Man_ON_OFF : Bool;
   //    END_STRUCT;
   //    Param : Struct
   //       SP_Level_LL : Real;
   //       SP_Level_ML : Real;
   //       SP_Level_HL : Real;
   //       SP_Temp_Prepar : Real;
   //       SP_Temp_Process : Real;
   //       SP_PumpSpeed : Real;
   //       L_Hi_Lim : Real;
   //       L_Lo_Lim : Real;
   //       L_Hys : Real;
   //       T_Hi_Lim : Real;
   //       T_Lo_Lim : Real;
   //       T_Hys : Real;
   //       CIP_Ret_ON_SP : Real;
   //       CIP_Ret_OFF_SP : Real;
   //    END_STRUCT;
   //    State : Struct
   //       Tank_LL : Bool;
   //       Tank_ML : Bool;
   //       Tank_HL : Bool;
   //       Temp_Preheat_OK : Bool;
   //       Temp_Process_OK : Bool;
   //       Tank_Heating : Bool;
   //       "Tank is Ready" : Bool;
   //       "Tank in transfer" : Bool;
   //       Enable_WHT_Mode : Bool;
   //       Enable_Ready : Bool;
   //       Ready_for_Mix : Bool;
   //       "CIP Request Enable" : Bool;
   //       "Tank in CIP" : Bool;
   //       CIP_Request_OK : Bool;
   //       CIP_ReturnON : Bool;
   //       HWT_Status : Int;
   //       Temp_Actual : Real;
   //    END_STRUCT;
   //    L_Hys_Abs : Real;
   //    T_Hys_Abs : Real;
   //    Hys_Level_HL : Real;
   //    Hys_Level_ML : Real;
   //    Hys_Level_LL : Real;
   //    "Hys SP_SP_Prepar" : Real;
   //    "Hys SP_SP_Process" : Real;
   //    "Hys SP_SP_" : Real;
   //    alwaysON : Bool;
   //    r : Struct
   //       PosE1 : Bool;
   //       PosE2 : Bool;
   //       PosE3 : Bool;
   //       PosE4 : Bool;
   //       PosE5 : Bool;
   //       PosE6 : Bool;
   //       PosE7 : Bool;
   //       PosE8 : Bool;
   //       PosE9 : Bool;
   //       PosE10 : Bool;
   //       PosE11 : Bool;
   //       PosE12 : Bool;
   //       PosE13 : Bool;
   //       PosE14 : Bool;
   //       PosE15 : Bool;
   //       PosE16 : Bool;
   //       PosE17 : Bool;
   //       PosE18 : Bool;
   //       PosE19 : Bool;
   //       PosE20 : Bool;
   //       PosE21 : Bool;
   //       PosE22 : Bool;
   //       PosE23 : Bool;
   //       PosE24 : Bool;
   //       PosE25 : Bool;
   //       PosE26 : Bool;
   //       PosE27 : Bool;
   //       PosE28 : Bool;
   //       PosE29 : Bool;
   //       PosE30 : Bool;
   //       PosE31 : Bool;
   //       PosE32 : Bool;
   //    END_STRUCT;
   //    Actuator : Struct
   //       AV_Inlet : Bool;
   //       AV_Return : Bool;
   //       CV_Steam : Bool;
   //       Pump : Bool;
   //    END_STRUCT;
   //    r_Pump : Bool;
   //    r_PumpTim { S7_SetPoint := 'True'} : IEC_TIMER;
   //    Alarm : Word;
   //    Event : Word;
   // END_VAR
BEGIN
END_DATA_BLOCK
